  MoveL 696 to (-315.68, 55.52, -14.28) mm, rotated rx -179.9 ry 0 rz -90 deg; joints [13.027, -91.875, 133.091, -160.309, 41.97, 165.528]
  MoveL 697 to (-315.68, 55.53, -297.96) mm, rotated rx -179.9 ry 0 rz -90 deg; joints [10.215, -74.026, 113.034, -163.714, 39.206, 167.625]
  MoveC 698 to (-314.55, 55.52, -300.68) mm, rotated rx -179.9 ry 0 rz -90 deg; joints [10.243, -73.85, 112.805, -163.654, 39.161, 167.569] to (-311.82, 55.53, -301.81) mm, rotated rx -179.9 ry 0 rz -90 deg; joints [10.35, -73.753, 112.677, -163.476, 39.155, 167.427]
  MoveL 699 to (-311.82, 55.53, -301.81) mm, rotated rx -179.9 ry 0 rz -90 deg; joints [10.35, -73.753, 112.677, -163.476, 39.155, 167.427]
  MoveL 700 to (311.82, 55.52, -301.81) mm, rotated rx -179.9 ry 0 rz -90 deg; joints [33.565, -59.232, 91.443, -127.903, 44.47, 138.323]
  MoveC 701 to (314.55, 55.52, -300.68) mm, rotated rx -179.9 ry 0 rz -90 deg; joints [33.672, -59.197, 91.385, -127.772, 44.528, 138.219] to (315.68, 55.52, -297.96) mm, rotated rx -179.9 ry 0 rz -90 deg; joints [33.762, -59.301, 91.545, -127.721, 44.622, 138.214]
  MoveL 702 to (315.68, 55.53, -297.96) mm, rotated rx -179.9 ry 0 rz -90 deg; joints [33.762, -59.301, 91.545, -127.721, 44.622, 138.214]
  MoveL 703 to (315.68, 55.53, -141.98) mm, rotated rx -179.9 ry 0 rz -90 deg; joints [37.25, -67.192, 103.214, -126.934, 49.209, 139.929]
  MoveC 704 to (314.4, 55.52, -137.76) mm, rotated rx -179.9 ry 0 rz -90 deg; joints [37.312, -67.444, 103.572, -126.944, 49.312, 140] to (311, 55.53, -134.96) mm, rotated rx -179.9 ry 0 rz -90 deg; joints [37.272, -67.705, 103.944, -127.061, 49.353, 140.143]
  MoveL 705 to (311, 55.53, -134.96) mm, rotated rx -179.9 ry 0 rz -90 deg; joints [37.272, -67.705, 103.944, -127.061, 49.353, 140.143]
  MoveC 706 to (307.59, 55.53, -132.16) mm, rotated rx -179.9 ry 0 rz -90 deg; joints [37.231, -67.966, 104.315, -127.177, 49.393, 140.284] to (306.32, 55.52, -127.94) mm, rotated rx -179.9 ry 0 rz -90 deg; joints [37.294, -68.219, 104.669, -127.184, 49.495, 140.351]
  MoveL 707 to (306.31, 55.53, -127.94) mm, rotated rx -179.9 ry 0 rz -90 deg; joints [37.294, -68.219, 104.669, -127.184, 49.495, 140.351]
  MoveL 708 to (306.32, 55.53, -23.64) mm, rotated rx -179.9 ry 0 rz -90 deg; joints [40.023, -73.194, 111.401, -125.63, 52.284, 140.513]
  MoveC 709 to (305.19, 55.52, -20.92) mm, rotated rx -179.9 ry 0 rz -90 deg; joints [40.061, -73.365, 111.626, -125.627, 52.34, 140.546] to (302.46, 55.53, -19.79) mm, rotated rx -179.9 ry 0 rz -90 deg; joints [40.003, -73.525, 111.837, -125.716, 52.333, 140.633]
  MoveL 710 to (302.46, 55.52, -19.79) mm, rotated rx -179.9 ry 0 rz -90 deg; joints [40.003, -73.525, 111.837, -125.716, 52.333, 140.633]
  MoveL 711 to (-302.46, 55.52, -19.79) mm, rotated rx -179.9 ry 0 rz -90 deg; joints [13.666, -91.295, 132.533, -159.397, 42.156, 164.867]
  MoveC 712 to (-305.19, 55.53, -20.92) mm, rotated rx -179.9 ry 0 rz -90 deg; joints [13.506, -91.263, 132.504, -159.629, 42.117, 165.037] to (-306.32, 55.53, -23.64) mm, rotated rx -179.9 ry 0 rz -90 deg; joints [13.41, -91.098, 132.348, -159.769, 42.099, 165.141]
  MoveL 713 to (-306.31, 55.53, -23.64) mm, rotated rx -179.9 ry 0 rz -90 deg; joints [13.41, -91.098, 132.348, -159.769, 42.099, 165.141]
  MoveL 714 to (-306.32, 55.52, -288.59) mm, rotated rx -179.9 ry 0 rz -90 deg; joints [10.693, -74.485, 113.625, -163.024, 39.438, 167.123]
  MoveC 715 to (-305.19, 55.53, -291.32) mm, rotated rx -179.9 ry 0 rz -90 deg; joints [10.72, -74.309, 113.397, -162.965, 39.394, 167.068] to (-302.46, 55.52, -292.45) mm, rotated rx -179.9 ry 0 rz -90 deg; joints [10.827, -74.211, 113.268, -162.789, 39.39, 166.928]
  MoveL 716 to (-302.46, 55.52, -292.45) mm, rotated rx -179.9 ry 0 rz -90 deg; joints [10.827, -74.211, 113.268, -162.789, 39.39, 166.928]
  MoveL 717 to (302.46, 55.52, -292.45) mm, rotated rx -179.9 ry 0 rz -90 deg; joints [33.468, -60.052, 92.711, -128.364, 44.683, 138.897]
  MoveC 718 to (305.19, 55.53, -291.32) mm, rotated rx -179.9 ry 0 rz -90 deg; joints [33.576, -60.017, 92.655, -128.232, 44.741, 138.794] to (306.32, 55.53, -288.59) mm, rotated rx -179.9 ry 0 rz -90 deg; joints [33.667, -60.121, 92.813, -128.178, 44.834, 138.786]
  MoveL 719 to (306.31, 55.53, -288.59) mm, rotated rx -179.9 ry 0 rz -90 deg; joints [33.667, -60.121, 92.813, -128.178, 44.834, 138.786]
  MoveL 720 to (306.31, 55.53, -127.94) mm, rotated rx -179.9 ry 0 rz -90 deg; joints [37.294, -68.219, 104.669, -127.184, 49.495, 140.351]
  MoveC 721 to (305.04, 55.52, -123.72) mm, rotated rx -179.9 ry 0 rz -90 deg; joints [37.357, -68.47, 105.022, -127.189, 49.596, 140.417] to (301.63, 55.53, -120.92) mm, rotated rx -179.9 ry 0 rz -90 deg; joints [37.316, -68.731, 105.389, -127.302, 49.634, 140.554]
  MoveL 722 to (301.63, 55.52, -120.92) mm, rotated rx -179.9 ry 0 rz -90 deg; joints [37.316, -68.731, 105.389, -127.302, 49.634, 140.554]
  MoveC 723 to (298.23, 55.53, -118.11) mm, rotated rx -179.9 ry 0 rz -90 deg; joints [37.275, -68.992, 105.754, -127.414, 49.672, 140.689] to (296.95, 55.53, -113.9) mm, rotated rx -179.9 ry 0 rz -90 deg; joints [37.338, -69.244, 106.104, -127.415, 49.772, 140.751]
  MoveL 724 to (296.95, 55.53, -113.9) mm, rotated rx -179.9 ry 0 rz -90 deg; joints [37.338, -69.244, 106.104, -127.415, 49.772, 140.751]
  MoveL 725 to (296.95, 55.53, -33) mm, rotated rx -179.9 ry 0 rz -90 deg; joints [39.455, -73.116, 111.311, -126.178, 51.915, 140.832]
  MoveC 726 to (295.82, 55.53, -30.28) mm, rotated rx -179.9 ry 0 rz -90 deg; joints [39.492, -73.288, 111.537, -126.175, 51.971, 140.866] to (293.1, 55.52, -29.15) mm, rotated rx -179.9 ry 0 rz -90 deg; joints [39.433, -73.446, 111.747, -126.267, 51.964, 140.954]
  MoveL 727 to (293.1, 55.53, -29.15) mm, rotated rx -179.9 ry 0 rz -90 deg; joints [39.433, -73.446, 111.747, -126.267, 51.964, 140.954]
  MoveL 728 to (-293.1, 55.52, -29.15) mm, rotated rx -179.9 ry 0 rz -90 deg; joints [14.039, -90.518, 131.781, -158.872, 42.278, 164.489]
  MoveC 729 to (-295.82, 55.52, -30.28) mm, rotated rx -179.9 ry 0 rz -90 deg; joints [13.88, -90.488, 131.753, -159.1, 42.238, 164.656] to (-296.95, 55.52, -33) mm, rotated rx -179.9 ry 0 rz -90 deg; joints [13.785, -90.325, 131.595, -159.238, 42.218, 164.758]
  MoveL 730 to (-296.95, 55.53, -33) mm, rotated rx -179.9 ry 0 rz -90 deg; joints [13.785, -90.325, 131.595, -159.238, 42.218, 164.758]
  MoveL 731 to (-296.95, 55.52, -279.23) mm, rotated rx -179.9 ry 0 rz -90 deg; joints [11.177, -74.94, 114.205, -162.331, 39.669, 166.62]
  MoveC 732 to (-295.82, 55.52, -281.95) mm, rotated rx -179.9 ry 0 rz -90 deg; joints [11.202, -74.763, 113.978, -162.274, 39.627, 166.566] to (-293.1, 55.53, -283.08) mm, rotated rx -179.9 ry 0 rz -90 deg; joints [11.31, -74.664, 113.848, -162.098, 39.624, 166.427]
  MoveL 733 to (-293.1, 55.53, -283.08) mm, rotated rx -179.9 ry 0 rz -90 deg; joints [11.31, -74.664, 113.848, -162.098, 39.624, 166.427]
  MoveL 734 to (293.1, 55.53, -283.08) mm, rotated rx -179.9 ry 0 rz -90 deg; joints [33.37, -60.867, 93.962, -128.813, 44.89, 139.454]
  MoveC 735 to (295.82, 55.53, -281.95) mm, rotated rx -179.9 ry 0 rz -90 deg; joints [33.478, -60.832, 93.907, -128.68, 44.948, 139.351] to (296.95, 55.53, -279.23) mm, rotated rx -179.9 ry 0 rz -90 deg; joints [33.57, -60.936, 94.063, -128.623, 45.041, 139.341]
  MoveL 736 to (296.95, 55.52, -279.23) mm, rotated rx -179.9 ry 0 rz -90 deg; joints [33.57, -60.936, 94.063, -128.623, 45.041, 139.341]
  MoveL 737 to (296.95, 55.53, -113.9) mm, rotated rx -179.9 ry 0 rz -90 deg; joints [37.338, -69.244, 106.104, -127.415, 49.772, 140.751]
  MoveC 738 to (295.67, 55.53, -109.68) mm, rotated rx -179.9 ry 0 rz -90 deg; joints [37.402, -69.495, 106.452, -127.416, 49.871, 140.81] to (292.27, 55.53, -106.87) mm, rotated rx -179.9 ry 0 rz -90 deg; joints [37.361, -69.756, 106.814, -127.525, 49.906, 140.942]
  MoveL 739 to (292.27, 55.52, -106.87) mm, rotated rx -179.9 ry 0 rz -90 deg; joints [37.361, -69.756, 106.814, -127.525, 49.907, 140.942]
  MoveC 740 to (288.87, 55.52, -104.07) mm, rotated rx -179.9 ry 0 rz -90 deg; joints [37.32, -70.017, 107.175, -127.634, 49.941, 141.072] to (287.59, 55.52, -99.85) mm, rotated rx -179.9 ry 0 rz -90 deg; joints [37.384, -70.268, 107.519, -127.63, 50.039, 141.127]
  MoveL 741 to (287.59, 55.52, -99.85) mm, rotated rx -179.9 ry 0 rz -90 deg; joints [37.384, -70.268, 107.519, -127.63, 50.039, 141.127]
  MoveL 742 to (287.59, 55.52, -42.37) mm, rotated rx -179.9 ry 0 rz -90 deg; joints [38.888, -73.029, 111.21, -126.728, 51.549, 141.155]
  MoveC 743 to (286.46, 55.52, -39.64) mm, rotated rx -179.9 ry 0 rz -90 deg; joints [38.924, -73.202, 111.438, -126.727, 51.604, 141.189] to (283.74, 55.52, -38.51) mm, rotated rx -179.9 ry 0 rz -90 deg; joints [38.864, -73.359, 111.647, -126.82, 51.597, 141.279]
  MoveL 744 to (283.74, 55.52, -38.51) mm, rotated rx -179.9 ry 0 rz -90 deg; joints [38.864, -73.359, 111.647, -126.82, 51.597, 141.279]
  MoveL 745 to (-283.74, 55.53, -38.51) mm, rotated rx -179.9 ry 0 rz -90 deg; joints [14.404, -89.745, 131.019, -158.355, 42.389, 164.116]
  MoveC 746 to (-286.46, 55.52, -39.64) mm, rotated rx -179.9 ry 0 rz -90 deg; joints [14.247, -89.716, 130.992, -158.58, 42.348, 164.28] to (-287.59, 55.53, -42.37) mm, rotated rx -179.9 ry 0 rz -90 deg; joints [14.152, -89.555, 130.834, -158.716, 42.325, 164.38]
  MoveL 747 to (-287.59, 55.52, -42.37) mm, rotated rx -179.9 ry 0 rz -90 deg; joints [14.152, -89.555, 130.834, -158.716, 42.325, 164.38]
  MoveL 748 to (-287.59, 55.52, -269.87) mm, rotated rx -179.9 ry 0 rz -90 deg; joints [11.666, -75.39, 114.775, -161.634, 39.901, 166.115]
  MoveC 749 to (-286.46, 55.52, -272.59) mm, rotated rx -179.9 ry 0 rz -90 deg; joints [11.69, -75.213, 114.548, -161.578, 39.86, 166.063] to (-283.74, 55.52, -273.72) mm, rotated rx -179.9 ry 0 rz -90 deg; joints [11.798, -75.111, 114.417, -161.404, 39.858, 165.925]
  MoveL 750 to (-283.74, 55.52, -273.72) mm, rotated rx -179.9 ry 0 rz -90 deg; joints [11.798, -75.111, 114.417, -161.404, 39.858, 165.925]
  MoveL 751 to (283.74, 55.52, -273.72) mm, rotated rx -179.9 ry 0 rz -90 deg; joints [33.27, -61.677, 95.196, -129.25, 45.092, 139.994]
  MoveC 752 to (286.46, 55.52, -272.59) mm, rotated rx -179.9 ry 0 rz -90 deg; joints [33.379, -61.643, 95.142, -129.116, 45.15, 139.891] to (287.59, 55.52, -269.87) mm, rotated rx -179.9 ry 0 rz -90 deg; joints [33.472, -61.746, 95.296, -129.056, 45.242, 139.878]
  MoveL 753 to (287.59, 55.53, -269.87) mm, rotated rx -179.9 ry 0 rz -90 deg; joints [33.472, -61.746, 95.296, -129.056, 45.242, 139.878]
  MoveL 754 to (287.59, 55.52, -99.85) mm, rotated rx -179.9 ry 0 rz -90 deg; joints [37.384, -70.268, 107.519, -127.63, 50.039, 141.127]
  MoveC 755 to (286.31, 55.53, -95.63) mm, rotated rx -179.9 ry 0 rz -90 deg; joints [37.449, -70.519, 107.863, -127.626, 50.136, 141.181] to (282.91, 55.52, -92.83) mm, rotated rx -179.9 ry 0 rz -90 deg; joints [37.407, -70.78, 108.22, -127.732, 50.169, 141.307]
  MoveL 756 to (282.91, 55.52, -92.83) mm, rotated rx -179.9 ry 0 rz -90 deg; joints [37.407, -70.78, 108.22, -127.732, 50.169, 141.307]
  MoveC 757 to (279.5, 55.52, -90.03) mm, rotated rx -179.9 ry 0 rz -90 deg; joints [37.366, -71.041, 108.576, -127.837, 50.201, 141.432] to (278.23, 55.52, -85.81) mm, rotated rx -179.9 ry 0 rz -90 deg; joints [37.431, -71.292, 108.916, -127.829, 50.296, 141.481]
  MoveL 758 to (278.23, 55.53, -85.81) mm, rotated rx -179.9 ry 0 rz -90 deg; joints [37.431, -71.292, 108.916, -127.829, 50.296, 141.481]
  MoveL 759 to (278.23, 55.53, -51.73) mm, rotated rx -179.9 ry 0 rz -90 deg; joints [38.323, -72.935, 111.099, -127.28, 51.183, 141.48]
  MoveC 760 to (277.1, 55.53, -49.01) mm, rotated rx -179.9 ry 0 rz -90 deg; joints [38.357, -73.108, 111.327, -127.281, 51.238, 141.515] to (274.37, 55.52, -47.88) mm, rotated rx -179.9 ry 0 rz -90 deg; joints [38.296, -73.265, 111.535, -127.376, 51.231, 141.605]
  MoveL 761 to (274.37, 55.52, -47.88) mm, rotated rx -179.9 ry 0 rz -90 deg; joints [38.296, -73.265, 111.535, -127.376, 51.231, 141.605]
  MoveL 762 to (-274.37, 55.52, -47.88) mm, rotated rx -179.9 ry 0 rz -90 deg; joints [14.762, -88.975, 130.248, -157.846, 42.489, 163.746]
  MoveC 763 to (-277.1, 55.52, -49.01) mm, rotated rx -179.9 ry 0 rz -90 deg; joints [14.606, -88.947, 130.222, -158.068, 42.447, 163.908] to (-278.23, 55.52, -51.73) mm, rotated rx -179.9 ry 0 rz -90 deg; joints [14.512, -88.789, 130.064, -158.202, 42.42, 164.005]
  MoveL 764 to (-278.23, 55.52, -51.73) mm, rotated rx -179.9 ry 0 rz -90 deg; joints [14.512, -88.789, 130.064, -158.202, 42.42, 164.005]
  MoveL 765 to (-278.23, 55.52, -260.51) mm, rotated rx -179.9 ry 0 rz -90 deg; joints [12.16, -75.835, 115.335, -160.932, 40.132, 165.61]
  MoveC 766 to (-277.1, 55.52, -263.23) mm, rotated rx -179.9 ry 0 rz -90 deg; joints [12.184, -75.657, 115.109, -160.879, 40.092, 165.559] to (-274.37, 55.52, -264.36) mm, rotated rx -179.9 ry 0 rz -90 deg; joints [12.292, -75.554, 114.977, -160.705, 40.092, 165.422]
  MoveL 767 to (-274.37, 55.52, -264.36) mm, rotated rx -179.9 ry 0 rz -90 deg; joints [12.292, -75.554, 114.977, -160.705, 40.092, 165.422]
  MoveL 768 to (274.37, 55.52, -264.36) mm, rotated rx -179.9 ry 0 rz -90 deg; joints [33.168, -62.482, 96.413, -129.675, 45.289, 140.518]
  MoveC 769 to (277.1, 55.52, -263.23) mm, rotated rx -179.9 ry 0 rz -90 deg; joints [33.279, -62.449, 96.36, -129.541, 45.347, 140.415] to (278.23, 55.52, -260.51) mm, rotated rx -179.9 ry 0 rz -90 deg; joints [33.372, -62.552, 96.513, -129.479, 45.438, 140.4]
  MoveL 770 to (278.23, 55.52, -260.51) mm, rotated rx -179.9 ry 0 rz -90 deg; joints [33.372, -62.552, 96.513, -129.479, 45.438, 140.4]
  MoveL 771 to (278.23, 55.53, -85.81) mm, rotated rx -179.9 ry 0 rz -90 deg; joints [37.431, -71.292, 108.916, -127.829, 50.296, 141.481]
  MoveC 772 to (276.95, 55.52, -81.59) mm, rotated rx -179.9 ry 0 rz -90 deg; joints [37.497, -71.544, 109.255, -127.819, 50.391, 141.529] to (273.55, 55.52, -78.79) mm, rotated rx -179.9 ry 0 rz -90 deg; joints [37.455, -71.805, 109.608, -127.922, 50.421, 141.65]
  MoveL 773 to (273.55, 55.52, -78.79) mm, rotated rx -179.9 ry 0 rz -90 deg; joints [37.455, -71.805, 109.608, -127.922, 50.421, 141.65]
  MoveC 774 to (270.14, 55.52, -75.98) mm, rotated rx -179.9 ry 0 rz -90 deg; joints [37.413, -72.065, 109.959, -128.024, 50.451, 141.769] to (268.86, 55.53, -71.76) mm, rotated rx -179.9 ry 0 rz -90 deg; joints [37.479, -72.317, 110.295, -128.011, 50.544, 141.813]
  MoveL 775 to (268.86, 55.53, -71.76) mm, rotated rx -179.9 ry 0 rz -90 deg; joints [37.479, -72.317, 110.295, -128.011, 50.544, 141.813]
  MoveL 776 to (268.86, 55.52, -61.09) mm, rotated rx -179.9 ry 0 rz -90 deg; joints [37.758, -72.834, 110.977, -127.835, 50.819, 141.807]
  MoveC 777 to (267.74, 55.53, -58.37) mm, rotated rx -179.9 ry 0 rz -90 deg; joints [37.792, -73.007, 111.206, -127.837, 50.874, 141.843] to (265.01, 55.53, -57.24) mm, rotated rx -179.9 ry 0 rz -90 deg; joints [37.729, -73.163, 111.413, -127.934, 50.867, 141.935]
  MoveL 778 to (265.01, 55.52, -57.24) mm, rotated rx -179.9 ry 0 rz -90 deg; joints [37.729, -73.163, 111.413, -127.934, 50.867, 141.935]
  MoveL 779 to (-265.01, 55.53, -57.24) mm, rotated rx -179.9 ry 0 rz -90 deg; joints [15.112, -88.208, 129.468, -157.345, 42.577, 163.379]
  MoveC 780 to (-267.74, 55.52, -58.37) mm, rotated rx -179.9 ry 0 rz -90 deg; joints [14.958, -88.182, 129.443, -157.563, 42.534, 163.538] to (-268.86, 55.53, -61.09) mm, rotated rx -179.9 ry 0 rz -90 deg; joints [14.863, -88.025, 129.284, -157.696, 42.505, 163.634]
  MoveL 781 to (-268.86, 55.52, -61.09) mm, rotated rx -179.9 ry 0 rz -90 deg; joints [14.863, -88.025, 129.284, -157.696, 42.505, 163.634]
  MoveL 782 to (-268.86, 55.52, -251.14) mm, rotated rx -179.9 ry 0 rz -90 deg; joints [12.661, -76.274, 115.884, -160.227, 40.363, 165.104]
  MoveC 783 to (-267.74, 55.53, -253.87) mm, rotated rx -179.9 ry 0 rz -90 deg; joints [12.683, -76.096, 115.658, -160.175, 40.325, 165.054] to (-265.01, 55.52, -255) mm, rotated rx -179.9 ry 0 rz -90 deg; joints [12.791, -75.992, 115.525, -160.003, 40.326, 164.918]
  MoveL 784 to (-265.01, 55.53, -255) mm, rotated rx -179.9 ry 0 rz -90 deg; joints [12.791, -75.992, 115.525, -160.003, 40.326, 164.918]
  MoveL 785 to (265.01, 55.52, -255) mm, rotated rx -179.9 ry 0 rz -90 deg; joints [33.065, -63.284, 97.615, -130.09, 45.479, 141.026]
  MoveC 786 to (267.74, 55.52, -253.87) mm, rotated rx -179.9 ry 0 rz -90 deg; joints [33.176, -63.251, 97.563, -129.955, 45.538, 140.923] to (268.86, 55.52, -251.14) mm, rotated rx -179.9 ry 0 rz -90 deg; joints [33.27, -63.354, 97.714, -129.89, 45.628, 140.906]
  MoveL 787 to (268.86, 55.52, -251.14) mm, rotated rx -179.9 ry 0 rz -90 deg; joints [33.27, -63.354, 97.714, -129.89, 45.628, 140.906]
  MoveL 788 to (268.86, 55.53, -71.76) mm, rotated rx -179.9 ry 0 rz -90 deg; joints [37.479, -72.317, 110.295, -128.011, 50.544, 141.813]
  MoveC 789 to (266.09, 55.52, -66.2) mm, rotated rx -179.9 ry 0 rz -90 deg; joints [37.53, -72.689, 110.789, -128.038, 50.651, 141.906] to (259.98, 55.53, -65.06) mm, rotated rx -179.9 ry 0 rz -90 deg; joints [37.352, -72.969, 111.165, -128.281, 50.601, 142.116]
  MoveL 790 to (259.98, 55.53, -65.06) mm, rotated rx -179.9 ry 0 rz -90 deg; joints [37.352, -72.969, 111.165, -128.281, 50.601, 142.116]
  MoveC 791 to (254.53, 55.52, -66.22) mm, rotated rx -179.9 ry 0 rz -90 deg; joints [37.136, -73.112, 111.361, -128.536, 50.499, 142.305] to (248.97, 55.53, -66.6) mm, rotated rx -179.9 ry 0 rz -90 deg; joints [36.934, -73.296, 111.608, -128.783, 50.416, 142.498]
  MoveL 792 to (248.97, 55.53, -66.6) mm, rotated rx -179.9 ry 0 rz -90 deg; joints [36.934, -73.296, 111.608, -128.783, 50.416, 142.498]
  MoveL 793 to (-255.65, 55.53, -66.6) mm, rotated rx -179.9 ry 0 rz -90 deg; joints [15.454, -87.444, 128.679, -156.85, 42.654, 163.014]
  MoveC 794 to (-258.37, 55.53, -67.73) mm, rotated rx -179.9 ry 0 rz -90 deg; joints [15.302, -87.42, 128.656, -157.066, 42.61, 163.171] to (-259.5, 55.52, -70.46) mm, rotated rx -179.9 ry 0 rz -90 deg; joints [15.208, -87.265, 128.496, -157.197, 42.578, 163.264]
  MoveL 795 to (-259.5, 55.52, -70.46) mm, rotated rx -179.9 ry 0 rz -90 deg; joints [15.208, -87.265, 128.496, -157.197, 42.578, 163.264]
  MoveL 796 to (-259.5, 55.52, -241.78) mm, rotated rx -179.9 ry 0 rz -90 deg; joints [13.166, -76.708, 116.422, -159.518, 40.595, 164.596]
  MoveC 797 to (-258.37, 55.53, -244.5) mm, rotated rx -179.9 ry 0 rz -90 deg; joints [13.188, -76.529, 116.198, -159.468, 40.558, 164.548] to (-255.65, 55.53, -245.63) mm, rotated rx -179.9 ry 0 rz -90 deg; joints [13.295, -76.424, 116.064, -159.297, 40.561, 164.413]
  MoveL 798 to (-255.65, 55.53, -245.63) mm, rotated rx -179.9 ry 0 rz -90 deg; joints [13.295, -76.424, 116.064, -159.297, 40.561, 164.413]
  MoveL 799 to (255.65, 55.52, -245.63) mm, rotated rx -179.9 ry 0 rz -90 deg; joints [32.959, -64.082, 98.801, -130.495, 45.664, 141.519]
  MoveC 800 to (258.37, 55.53, -244.5) mm, rotated rx -179.9 ry 0 rz -90 deg; joints [33.072, -64.05, 98.751, -130.359, 45.723, 141.416] to (259.5, 55.52, -241.78) mm, rotated rx -179.9 ry 0 rz -90 deg; joints [33.166, -64.153, 98.901, -130.291, 45.812, 141.396]
  MoveL 801 to (259.5, 55.52, -241.78) mm, rotated rx -179.9 ry 0 rz -90 deg; joints [33.166, -64.153, 98.901, -130.291, 45.812, 141.396]
  MoveL 802 to (259.5, 55.53, -70.46) mm, rotated rx -179.9 ry 0 rz -90 deg; joints [37.195, -72.724, 110.844, -128.392, 50.456, 142.137]
  MoveC 803 to (258.37, 55.53, -67.73) mm, rotated rx -179.9 ry 0 rz -90 deg; joints [37.228, -72.898, 111.074, -128.395, 50.511, 142.174] to (255.65, 55.52, -66.6) mm, rotated rx -179.9 ry 0 rz -90 deg; joints [37.164, -73.052, 111.281, -128.494, 50.504, 142.267]
  MoveL 804 to (255.65, 55.52, -66.6) mm, rotated rx -179.9 ry 0 rz -90 deg; joints [37.164, -73.052, 111.281, -128.494, 50.504, 142.267]
  MoveL 805 to (248.97, 55.53, -66.6) mm, rotated rx -179.9 ry 0 rz -90 deg; joints [36.934, -73.296, 111.608, -128.783, 50.416, 142.498]
  MoveC 806 to (244.46, 55.52, -67.86) mm, rotated rx -179.9 ry 0 rz -90 deg; joints [36.746, -73.398, 111.746, -129, 50.324, 142.655] to (241.27, 55.52, -71.28) mm, rotated rx -179.9 ry 0 rz -90 deg; joints [36.547, -73.345, 111.682, -129.197, 50.195, 142.771]
  MoveL 807 to (241.27, 55.52, -71.28) mm, rotated rx -179.9 ry 0 rz -90 deg; joints [36.547, -73.345, 111.682, -129.197, 50.195, 142.771]
  MoveC 808 to (238.08, 55.52, -74.7) mm, rotated rx -179.9 ry 0 rz -90 deg; joints [36.349, -73.292, 111.616, -129.395, 50.067, 142.886] to (233.58, 55.53, -75.96) mm, rotated rx -179.9 ry 0 rz -90 deg; joints [36.16, -73.391, 111.75, -129.614, 49.975, 143.046]
  MoveL 809 to (233.58, 55.53, -75.96) mm, rotated rx -179.9 ry 0 rz -90 deg; joints [36.16, -73.391, 111.75, -129.614, 49.975, 143.046]
  MoveL 810 to (-246.29, 55.53, -75.96) mm, rotated rx -179.9 ry 0 rz -90 deg; joints [15.79, -86.684, 127.882, -156.362, 42.721, 162.651]
  MoveC 811 to (-249.01, 55.53, -77.09) mm, rotated rx -179.9 ry 0 rz -90 deg; joints [15.639, -86.66, 127.859, -156.575, 42.676, 162.805] to (-250.14, 55.52, -79.82) mm, rotated rx -179.9 ry 0 rz -90 deg; joints [15.545, -86.507, 127.699, -156.704, 42.641, 162.896]
  MoveL 812 to (-250.14, 55.53, -79.82) mm, rotated rx -179.9 ry 0 rz -90 deg; joints [15.545, -86.507, 127.699, -156.704, 42.641, 162.896]
  MoveL 813 to (-250.14, 55.52, -232.42) mm, rotated rx -179.9 ry 0 rz -90 deg; joints [13.677, -77.137, 116.95, -158.806, 40.828, 164.087]
  MoveC 814 to (-249.01, 55.53, -235.14) mm, rotated rx -179.9 ry 0 rz -90 deg; joints [13.698, -76.958, 116.727, -158.757, 40.792, 164.04] to (-246.29, 55.52, -236.27) mm, rotated rx -179.9 ry 0 rz -90 deg; joints [13.805, -76.851, 116.592, -158.588, 40.796, 163.907]
  MoveL 815 to (-246.29, 55.53, -236.27) mm, rotated rx -179.9 ry 0 rz -90 deg; joints [13.805, -76.851, 116.592, -158.588, 40.796, 163.907]
  MoveL 816 to (246.29, 55.53, -236.27) mm, rotated rx -179.9 ry 0 rz -90 deg; joints [32.852, -64.878, 99.973, -130.89, 45.843, 141.998]
  MoveC 817 to (249.01, 55.53, -235.14) mm, rotated rx -179.9 ry 0 rz -90 deg; joints [32.966, -64.846, 99.924, -130.754, 45.902, 141.895] to (250.14, 55.52, -232.42) mm, rotated rx -179.9 ry 0 rz -90 deg; joints [33.061, -64.949, 100.072, -130.683, 45.99, 141.873]
  MoveL 818 to (250.14, 55.53, -232.42) mm, rotated rx -179.9 ry 0 rz -90 deg; joints [33.061, -64.949, 100.072, -130.683, 45.99, 141.873]
  MoveL 819 to (250.14, 55.53, -79.82) mm, rotated rx -179.9 ry 0 rz -90 deg; joints [36.634, -72.607, 110.701, -128.951, 50.095, 142.47]
  MoveC 820 to (249.01, 55.53, -77.09) mm, rotated rx -179.9 ry 0 rz -90 deg; joints [36.665, -72.781, 110.932, -128.956, 50.15, 142.508] to (246.29, 55.53, -75.96) mm, rotated rx -179.9 ry 0 rz -90 deg; joints [36.6, -72.935, 111.137, -129.056, 50.143, 142.602]
  MoveL 821 to (246.29, 55.52, -75.96) mm, rotated rx -179.9 ry 0 rz -90 deg; joints [36.6, -72.934, 111.137, -129.056, 50.143, 142.602]
  MoveL 822 to (233.58, 55.53, -75.96) mm, rotated rx -179.9 ry 0 rz -90 deg; joints [36.16, -73.391, 111.75, -129.614, 49.975, 143.046]
  MoveC 823 to (229.36, 55.52, -77.24) mm, rotated rx -179.9 ry 0 rz -90 deg; joints [35.98, -73.478, 111.869, -129.822, 49.887, 143.195] to (226.56, 55.52, -80.65) mm, rotated rx -179.9 ry 0 rz -90 deg; joints [35.795, -73.409, 111.782, -130.003, 49.765, 143.299]
  MoveL 824 to (226.56, 55.52, -80.65) mm, rotated rx -179.9 ry 0 rz -90 deg; joints [35.795, -73.409, 111.782, -130.003, 49.765, 143.299]
  MoveC 825 to (223.75, 55.53, -84.05) mm, rotated rx -179.9 ry 0 rz -90 deg; joints [35.611, -73.338, 111.694, -130.185, 49.642, 143.403] to (219.54, 55.53, -85.33) mm, rotated rx -179.9 ry 0 rz -90 deg; joints [35.431, -73.423, 111.81, -130.395, 49.555, 143.554]
  MoveL 826 to (219.54, 55.53, -85.33) mm, rotated rx -179.9 ry 0 rz -90 deg; joints [35.431, -73.423, 111.81, -130.395, 49.555, 143.554]
  MoveL 827 to (-236.92, 55.52, -85.33) mm, rotated rx -179.9 ry 0 rz -90 deg; joints [16.119, -85.926, 127.075, -155.88, 42.776, 162.289]
  MoveC 828 to (-239.65, 55.53, -86.46) mm, rotated rx -179.9 ry 0 rz -90 deg; joints [15.969, -85.904, 127.053, -156.089, 42.731, 162.44] to (-240.78, 55.52, -89.18) mm, rotated rx -179.9 ry 0 rz -90 deg; joints [15.876, -85.753, 126.893, -156.217, 42.694, 162.53]
  MoveL 829 to (-240.78, 55.52, -89.18) mm, rotated rx -179.9 ry 0 rz -90 deg; joints [15.876, -85.753, 126.893, -156.217, 42.694, 162.53]
  MoveL 830 to (-240.78, 55.52, -223.05) mm, rotated rx -179.9 ry 0 rz -90 deg; joints [14.194, -77.561, 117.468, -158.089, 41.061, 163.577]
  MoveC 831 to (-239.65, 55.52, -225.78) mm, rotated rx -179.9 ry 0 rz -90 deg; joints [14.213, -77.381, 117.245, -158.043, 41.027, 163.532] to (-236.92, 55.52, -226.91) mm, rotated rx -179.9 ry 0 rz -90 deg; joints [14.321, -77.272, 117.109, -157.874, 41.033, 163.4]
  MoveL 832 to (-236.92, 55.52, -226.91) mm, rotated rx -179.9 ry 0 rz -90 deg; joints [14.321, -77.272, 117.109, -157.874, 41.033, 163.4]
  MoveL 833 to (236.92, 55.52, -226.91) mm, rotated rx -179.9 ry 0 rz -90 deg; joints [32.743, -65.671, 101.131, -131.277, 46.016, 142.463]
  MoveC 834 to (239.65, 55.53, -225.78) mm, rotated rx -179.9 ry 0 rz -90 deg; joints [32.857, -65.639, 101.083, -131.139, 46.075, 142.36] to (240.78, 55.53, -223.05) mm, rotated rx -179.9 ry 0 rz -90 deg; joints [32.953, -65.742, 101.23, -131.066, 46.163, 142.335]
  MoveL 835 to (240.78, 55.53, -223.05) mm, rotated rx -179.9 ry 0 rz -90 deg; joints [32.953, -65.742, 101.23, -131.066, 46.163, 142.335]
  MoveL 836 to (240.78, 55.53, -89.18) mm, rotated rx -179.9 ry 0 rz -90 deg; joints [36.074, -72.481, 110.547, -129.512, 49.736, 142.805]
  MoveC 837 to (239.65, 55.52, -86.46) mm, rotated rx -179.9 ry 0 rz -90 deg; joints [36.104, -72.656, 110.779, -129.518, 49.79, 142.843] to (236.92, 55.52, -85.33) mm, rotated rx -179.9 ry 0 rz -90 deg; joints [36.038, -72.809, 110.984, -129.621, 49.783, 142.939]
  MoveL 838 to (236.92, 55.52, -85.33) mm, rotated rx -179.9 ry 0 rz -90 deg; joints [36.038, -72.809, 110.984, -129.621, 49.783, 142.939]
  MoveL 839 to (219.54, 55.53, -85.33) mm, rotated rx -179.9 ry 0 rz -90 deg; joints [35.431, -73.423, 111.81, -130.395, 49.555, 143.554]
  MoveC 840 to (215.32, 55.52, -86.61) mm, rotated rx -179.9 ry 0 rz -90 deg; joints [35.25, -73.507, 111.924, -130.605, 49.467, 143.705] to (212.51, 55.52, -90.01) mm, rotated rx -179.9 ry 0 rz -90 deg; joints [35.066, -73.435, 111.833, -130.788, 49.345, 143.81]
  MoveL 841 to (212.51, 55.52, -90.01) mm, rotated rx -179.9 ry 0 rz -90 deg; joints [35.066, -73.435, 111.833, -130.788, 49.345, 143.81]
  MoveC 842 to (209.71, 55.53, -93.41) mm, rotated rx -179.9 ry 0 rz -90 deg; joints [34.883, -73.361, 111.74, -130.97, 49.224, 143.915] to (205.49, 55.53, -94.69) mm, rotated rx -179.9 ry 0 rz -90 deg; joints [34.701, -73.443, 111.852, -131.183, 49.136, 144.068]
  MoveL 843 to (205.49, 55.53, -94.69) mm, rotated rx -179.9 ry 0 rz -90 deg; joints [34.701, -73.443, 111.852, -131.183, 49.136, 144.068]
  MoveL 844 to (-227.56, 55.52, -94.69) mm, rotated rx -179.9 ry 0 rz -90 deg; joints [16.44, -85.171, 126.26, -155.403, 42.821, 161.927]
  MoveC 845 to (-230.29, 55.52, -95.82) mm, rotated rx -179.9 ry 0 rz -90 deg; joints [16.292, -85.15, 126.239, -155.61, 42.775, 162.076] to (-231.41, 55.53, -98.54) mm, rotated rx -179.9 ry 0 rz -90 deg; joints [16.199, -85, 126.078, -155.735, 42.736, 162.164]
  MoveL 846 to (-231.41, 55.52, -98.54) mm, rotated rx -179.9 ry 0 rz -90 deg; joints [16.199, -85, 126.078, -155.735, 42.736, 162.164]
  MoveL 847 to (-231.41, 55.53, -213.69) mm, rotated rx -179.9 ry 0 rz -90 deg; joints [14.717, -77.979, 117.976, -157.369, 41.296, 163.065]
  MoveC 848 to (-230.29, 55.52, -216.42) mm, rotated rx -179.9 ry 0 rz -90 deg; joints [14.735, -77.798, 117.753, -157.324, 41.263, 163.022] to (-227.56, 55.52, -217.54) mm, rotated rx -179.9 ry 0 rz -90 deg; joints [14.842, -77.688, 117.616, -157.157, 41.27, 162.891]
  MoveL 849 to (-227.56, 55.53, -217.55) mm, rotated rx -179.9 ry 0 rz -90 deg; joints [14.842, -77.688, 117.616, -157.157, 41.27, 162.891]
  MoveL 850 to (227.56, 55.53, -217.55) mm, rotated rx -179.9 ry 0 rz -90 deg; joints [32.632, -66.461, 102.275, -131.654, 46.182, 142.914]
  MoveC 851 to (230.29, 55.52, -216.42) mm, rotated rx -179.9 ry 0 rz -90 deg; joints [32.747, -66.43, 102.228, -131.515, 46.242, 142.811] to (231.41, 55.52, -213.69) mm, rotated rx -179.9 ry 0 rz -90 deg; joints [32.844, -66.533, 102.374, -131.44, 46.329, 142.784]
  MoveL 852 to (231.41, 55.52, -213.69) mm, rotated rx -179.9 ry 0 rz -90 deg; joints [32.844, -66.533, 102.374, -131.44, 46.329, 142.784]
  MoveL 853 to (231.41, 55.52, -98.54) mm, rotated rx -179.9 ry 0 rz -90 deg; joints [35.516, -72.349, 110.382, -130.075, 49.378, 143.142]
  MoveC 854 to (230.29, 55.52, -95.82) mm, rotated rx -179.9 ry 0 rz -90 deg; joints [35.544, -72.524, 110.615, -130.083, 49.432, 143.182] to (227.56, 55.53, -94.69) mm, rotated rx -179.9 ry 0 rz -90 deg; joints [35.478, -72.675, 110.819, -130.187, 49.425, 143.279]
  MoveL 855 to (227.56, 55.52, -94.69) mm, rotated rx -179.9 ry 0 rz -90 deg; joints [35.478, -72.675, 110.819, -130.187, 49.425, 143.279]
  MoveL 856 to (205.49, 55.53, -94.69) mm, rotated rx -179.9 ry 0 rz -90 deg; joints [34.701, -73.443, 111.852, -131.183, 49.136, 144.068]
  MoveC 857 to (201.27, 55.53, -95.97) mm, rotated rx -179.9 ry 0 rz -90 deg; joints [34.52, -73.524, 111.962, -131.396, 49.049, 144.222] to (198.47, 55.53, -99.37) mm, rotated rx -179.9 ry 0 rz -90 deg; joints [34.336, -73.448, 111.866, -131.58, 48.928, 144.328]
  MoveL 858 to (198.47, 55.52, -99.37) mm, rotated rx -179.9 ry 0 rz -90 deg; joints [34.336, -73.448, 111.866, -131.58, 48.928, 144.328]
  MoveC 859 to (195.67, 55.53, -102.78) mm, rotated rx -179.9 ry 0 rz -90 deg; joints [34.153, -73.371, 111.769, -131.764, 48.808, 144.435] to (191.45, 55.52, -104.05) mm, rotated rx -179.9 ry 0 rz -90 deg; joints [33.971, -73.449, 111.877, -131.979, 48.721, 144.59]
  MoveL 860 to (191.45, 55.52, -104.05) mm, rotated rx -179.9 ry 0 rz -90 deg; joints [33.971, -73.449, 111.877, -131.979, 48.721, 144.59]
  MoveL 861 to (-218.2, 55.53, -104.05) mm, rotated rx -179.9 ry 0 rz -90 deg; joints [16.756, -84.418, 125.435, -154.93, 42.856, 161.565]
  MoveC 862 to (-220.92, 55.53, -105.18) mm, rotated rx -179.9 ry 0 rz -90 deg; joints [16.609, -84.398, 125.415, -155.134, 42.809, 161.712] to (-222.05, 55.53, -107.91) mm, rotated rx -179.9 ry 0 rz -90 deg; joints [16.516, -84.25, 125.254, -155.258, 42.767, 161.798]
  MoveL 863 to (-222.05, 55.52, -107.91) mm, rotated rx -179.9 ry 0 rz -90 deg; joints [16.516, -84.25, 125.254, -155.258, 42.767, 161.798]
  MoveL 864 to (-222.05, 55.52, -204.33) mm, rotated rx -179.9 ry 0 rz -90 deg; joints [15.245, -78.391, 118.473, -156.645, 41.532, 162.553]
  MoveC 865 to (-220.92, 55.52, -207.05) mm, rotated rx -179.9 ry 0 rz -90 deg; joints [15.262, -78.21, 118.251, -156.602, 41.5, 162.511] to (-218.2, 55.53, -208.18) mm, rotated rx -179.9 ry 0 rz -90 deg; joints [15.369, -78.098, 118.113, -156.437, 41.508, 162.382]
  MoveL 866 to (-218.2, 55.53, -208.18) mm, rotated rx -179.9 ry 0 rz -90 deg; joints [15.369, -78.098, 118.113, -156.437, 41.508, 162.382]
  MoveL 867 to (218.2, 55.52, -208.18) mm, rotated rx -179.9 ry 0 rz -90 deg; joints [32.519, -67.249, 103.406, -132.023, 46.343, 143.352]
  MoveC 868 to (220.92, 55.53, -207.05) mm, rotated rx -179.9 ry 0 rz -90 deg; joints [32.635, -67.218, 103.36, -131.884, 46.402, 143.249] to (222.05, 55.52, -204.33) mm, rotated rx -179.9 ry 0 rz -90 deg; joints [32.733, -67.322, 103.505, -131.806, 46.489, 143.219]
  MoveL 869 to (222.05, 55.52, -204.33) mm, rotated rx -179.9 ry 0 rz -90 deg; joints [32.733, -67.322, 103.505, -131.806, 46.489, 143.219]
  MoveL 870 to (222.05, 55.53, -107.91) mm, rotated rx -179.9 ry 0 rz -90 deg; joints [34.959, -72.208, 110.207, -130.64, 49.021, 143.482]
  MoveC 871 to (220.92, 55.53, -105.18) mm, rotated rx -179.9 ry 0 rz -90 deg; joints [34.987, -72.384, 110.441, -130.649, 49.075, 143.523] to (218.2, 55.53, -104.05) mm, rotated rx -179.9 ry 0 rz -90 deg; joints [34.919, -72.534, 110.644, -130.755, 49.069, 143.621]
  MoveL 872 to (218.2, 55.53, -104.05) mm, rotated rx -179.9 ry 0 rz -90 deg; joints [34.919, -72.534, 110.644, -130.755, 49.069, 143.621]
  MoveL 873 to (191.45, 55.52, -104.05) mm, rotated rx -179.9 ry 0 rz -90 deg; joints [33.971, -73.449, 111.877, -131.979, 48.721, 144.59]
  MoveC 874 to (187.23, 55.52, -105.33) mm, rotated rx -179.9 ry 0 rz -90 deg; joints [33.789, -73.527, 111.982, -132.195, 48.634, 144.745] to (184.43, 55.52, -108.73) mm, rotated rx -179.9 ry 0 rz -90 deg; joints [33.606, -73.448, 111.882, -132.38, 48.514, 144.853]
  MoveL 875 to (184.43, 55.53, -108.73) mm, rotated rx -179.9 ry 0 rz -90 deg; joints [33.606, -73.448, 111.882, -132.38, 48.514, 144.853]
  MoveC 876 to (181.62, 55.52, -112.14) mm, rotated rx -179.9 ry 0 rz -90 deg; joints [33.424, -73.368, 111.781, -132.565, 48.394, 144.961] to (177.4, 55.52, -113.42) mm, rotated rx -179.9 ry 0 rz -90 deg; joints [33.241, -73.443, 111.884, -132.783, 48.307, 145.118]
  MoveL 877 to (177.4, 55.53, -113.42) mm, rotated rx -179.9 ry 0 rz -90 deg; joints [33.241, -73.443, 111.884, -132.783, 48.307, 145.118]
  MoveL 878 to (-208.84, 55.53, -113.42) mm, rotated rx -179.9 ry 0 rz -90 deg; joints [17.065, -83.668, 124.602, -154.462, 42.88, 161.203]
  MoveC 879 to (-211.56, 55.52, -114.54) mm, rotated rx -179.9 ry 0 rz -90 deg; joints [16.92, -83.649, 124.583, -154.664, 42.833, 161.348] to (-212.69, 55.53, -117.27) mm, rotated rx -179.9 ry 0 rz -90 deg; joints [16.827, -83.503, 124.421, -154.785, 42.789, 161.431]
  MoveL 880 to (-212.69, 55.53, -117.27) mm, rotated rx -179.9 ry 0 rz -90 deg; joints [16.827, -83.503, 124.421, -154.785, 42.789, 161.431]
  MoveL 881 to (-212.69, 55.53, -194.97) mm, rotated rx -179.9 ry 0 rz -90 deg; joints [15.778, -78.798, 118.959, -155.917, 41.769, 162.039]
  MoveC 882 to (-211.56, 55.52, -197.69) mm, rotated rx -179.9 ry 0 rz -90 deg; joints [15.794, -78.616, 118.739, -155.877, 41.739, 161.999] to (-208.84, 55.53, -198.82) mm, rotated rx -179.9 ry 0 rz -90 deg; joints [15.901, -78.503, 118.6, -155.712, 41.748, 161.871]
  MoveL 883 to (-208.84, 55.52, -198.82) mm, rotated rx -179.9 ry 0 rz -90 deg; joints [15.901, -78.503, 118.6, -155.712, 41.748, 161.871]
  MoveL 884 to (208.84, 55.53, -198.82) mm, rotated rx -179.9 ry 0 rz -90 deg; joints [32.404, -68.036, 104.525, -132.385, 46.497, 143.777]
  MoveC 885 to (211.56, 55.52, -197.69) mm, rotated rx -179.9 ry 0 rz -90 deg; joints [32.521, -68.006, 104.479, -132.244, 46.557, 143.674] to (212.69, 55.52, -194.97) mm, rotated rx -179.9 ry 0 rz -90 deg; joints [32.62, -68.109, 104.623, -132.164, 46.642, 143.642]
  MoveL 886 to (212.69, 55.53, -194.97) mm, rotated rx -179.9 ry 0 rz -90 deg; joints [32.62, -68.109, 104.623, -132.164, 46.642, 143.642]
  MoveL 887 to (212.69, 55.53, -117.27) mm, rotated rx -179.9 ry 0 rz -90 deg; joints [34.405, -72.06, 110.021, -131.206, 48.666, 143.825]
  MoveC 888 to (211.56, 55.52, -114.54) mm, rotated rx -179.9 ry 0 rz -90 deg; joints [34.431, -72.236, 110.256, -131.217, 48.72, 143.866] to (208.84, 55.52, -113.42) mm, rotated rx -179.9 ry 0 rz -90 deg; joints [34.363, -72.386, 110.458, -131.325, 48.714, 143.965]
  MoveL 889 to (208.84, 55.53, -113.42) mm, rotated rx -179.9 ry 0 rz -90 deg; joints [34.363, -72.386, 110.458, -131.325, 48.714, 143.965]
  MoveL 890 to (177.4, 55.53, -113.42) mm, rotated rx -179.9 ry 0 rz -90 deg; joints [33.241, -73.443, 111.884, -132.783, 48.307, 145.118]
  MoveC 891 to (173.18, 55.53, -114.69) mm, rotated rx -179.9 ry 0 rz -90 deg; joints [33.058, -73.517, 111.986, -133.002, 48.221, 145.276] to (170.38, 55.53, -118.1) mm, rotated rx -179.9 ry 0 rz -90 deg; joints [32.876, -73.435, 111.881, -133.188, 48.102, 145.385]
  MoveL 892 to (170.38, 55.52, -118.1) mm, rotated rx -179.9 ry 0 rz -90 deg; joints [32.876, -73.435, 111.881, -133.188, 48.102, 145.385]
  MoveC 893 to (167.58, 55.53, -121.5) mm, rotated rx -179.9 ry 0 rz -90 deg; joints [32.695, -73.352, 111.776, -133.373, 47.983, 145.494] to (163.36, 55.52, -122.78) mm, rotated rx -179.9 ry 0 rz -90 deg; joints [32.512, -73.424, 111.874, -133.594, 47.897, 145.653]
  MoveL 894 to (163.36, 55.52, -122.78) mm, rotated rx -179.9 ry 0 rz -90 deg; joints [32.512, -73.424, 111.874, -133.594, 47.897, 145.653]
  MoveL 895 to (-199.47, 55.52, -122.78) mm, rotated rx -179.9 ry 0 rz -90 deg; joints [17.368, -82.92, 123.76, -153.997, 42.895, 160.839]
  MoveC 896 to (-202.2, 55.53, -123.91) mm, rotated rx -179.9 ry 0 rz -90 deg; joints [17.224, -82.903, 123.742, -154.197, 42.847, 160.983] to (-203.33, 55.53, -126.63) mm, rotated rx -179.9 ry 0 rz -90 deg; joints [17.132, -82.758, 123.579, -154.317, 42.801, 161.064]
  MoveL 897 to (-203.33, 55.53, -126.63) mm, rotated rx -179.9 ry 0 rz -90 deg; joints [17.132, -82.758, 123.579, -154.317, 42.801, 161.064]
  MoveL 898 to (-203.33, 55.53, -185.6) mm, rotated rx -179.9 ry 0 rz -90 deg; joints [16.318, -79.199, 119.436, -155.186, 42.008, 161.524]
  MoveC 899 to (-202.2, 55.53, -188.33) mm, rotated rx -179.9 ry 0 rz -90 deg; joints [16.332, -79.016, 119.216, -155.147, 41.979, 161.486] to (-199.47, 55.53, -189.46) mm, rotated rx -179.9 ry 0 rz -90 deg; joints [16.439, -78.902, 119.076, -154.985, 41.99, 161.359]
  MoveL 900 to (-199.47, 55.53, -189.46) mm, rotated rx -179.9 ry 0 rz -90 deg; joints [16.439, -78.902, 119.076, -154.985, 41.99, 161.359]
  MoveL 901 to (199.47, 55.52, -189.46) mm, rotated rx -179.9 ry 0 rz -90 deg; joints [32.286, -68.821, 105.631, -132.739, 46.645, 144.19]
  MoveC 902 to (202.2, 55.52, -188.33) mm, rotated rx -179.9 ry 0 rz -90 deg; joints [32.405, -68.791, 105.586, -132.596, 46.705, 144.086] to (203.33, 55.52, -185.6) mm, rotated rx -179.9 ry 0 rz -90 deg; joints [32.504, -68.895, 105.729, -132.514, 46.789, 144.052]
  MoveL 903 to (203.33, 55.52, -185.6) mm, rotated rx -179.9 ry 0 rz -90 deg; joints [32.504, -68.895, 105.729, -132.514, 46.789, 144.052]
  MoveL 904 to (203.33, 55.52, -126.63) mm, rotated rx -179.9 ry 0 rz -90 deg; joints [33.852, -71.904, 109.824, -131.774, 48.312, 144.169]
  MoveC 905 to (202.2, 55.52, -123.91) mm, rotated rx -179.9 ry 0 rz -90 deg; joints [33.877, -72.08, 110.06, -131.787, 48.367, 144.211] to (199.47, 55.53, -122.78) mm, rotated rx -179.9 ry 0 rz -90 deg; joints [33.808, -72.229, 110.261, -131.896, 48.361, 144.312]
  MoveL 906 to (199.47, 55.53, -122.78) mm, rotated rx -179.9 ry 0 rz -90 deg; joints [33.808, -72.229, 110.261, -131.896, 48.361, 144.312]
  MoveL 907 to (163.36, 55.52, -122.78) mm, rotated rx -179.9 ry 0 rz -90 deg; joints [32.512, -73.424, 111.874, -133.594, 47.897, 145.653]
  MoveC 908 to (159.14, 55.53, -124.06) mm, rotated rx -179.9 ry 0 rz -90 deg; joints [32.328, -73.495, 111.971, -133.815, 47.811, 145.813] to (156.34, 55.53, -127.46) mm, rotated rx -179.9 ry 0 rz -90 deg; joints [32.147, -73.409, 111.863, -134.002, 47.693, 145.923]
  MoveL 909 to (156.34, 55.52, -127.46) mm, rotated rx -179.9 ry 0 rz -90 deg; joints [32.147, -73.409, 111.863, -134.002, 47.693, 145.923]
  MoveC 910 to (153.54, 55.52, -130.86) mm, rotated rx -179.9 ry 0 rz -90 deg; joints [31.966, -73.323, 111.753, -134.189, 47.575, 146.033] to (149.32, 55.53, -132.14) mm, rotated rx -179.9 ry 0 rz -90 deg; joints [31.782, -73.391, 111.847, -134.412, 47.49, 146.195]
  MoveL 911 to (149.32, 55.52, -132.14) mm, rotated rx -179.9 ry 0 rz -90 deg; joints [31.782, -73.391, 111.847, -134.412, 47.49, 146.195]
  MoveL 912 to (-190.11, 55.52, -132.14) mm, rotated rx -179.9 ry 0 rz -90 deg; joints [17.665, -82.174, 122.908, -153.536, 42.899, 160.475]
  MoveC 913 to (-192.84, 55.52, -133.27) mm, rotated rx -179.9 ry 0 rz -90 deg; joints [17.522, -82.158, 122.891, -153.733, 42.851, 160.616] to (-193.96, 55.53, -135.99) mm, rotated rx -179.9 ry 0 rz -90 deg; joints [17.43, -82.014, 122.728, -153.851, 42.803, 160.696]
  MoveL 914 to (-193.96, 55.53, -135.99) mm, rotated rx -179.9 ry 0 rz -90 deg; joints [17.43, -82.014, 122.728, -153.851, 42.803, 160.696]
  MoveL 915 to (-193.96, 55.52, -176.24) mm, rotated rx -179.9 ry 0 rz -90 deg; joints [16.862, -79.594, 119.902, -154.451, 42.249, 161.009]
  MoveC 916 to (-192.84, 55.53, -178.97) mm, rotated rx -179.9 ry 0 rz -90 deg; joints [16.876, -79.411, 119.682, -154.415, 42.221, 160.972] to (-190.11, 55.52, -180.09) mm, rotated rx -179.9 ry 0 rz -90 deg; joints [16.982, -79.294, 119.541, -154.254, 42.234, 160.847]
  MoveL 917 to (-190.11, 55.53, -180.09) mm, rotated rx -179.9 ry 0 rz -90 deg; joints [16.982, -79.294, 119.541, -154.254, 42.234, 160.847]
  MoveL 918 to (190.11, 55.52, -180.09) mm, rotated rx -179.9 ry 0 rz -90 deg; joints [32.167, -69.606, 106.725, -133.085, 46.785, 144.591]
  MoveC 919 to (192.84, 55.52, -178.97) mm, rotated rx -179.9 ry 0 rz -90 deg; joints [32.287, -69.576, 106.681, -132.942, 46.846, 144.487] to (193.96, 55.52, -176.24) mm, rotated rx -179.9 ry 0 rz -90 deg; joints [32.387, -69.68, 106.823, -132.857, 46.93, 144.451]
  MoveL 920 to (193.96, 55.52, -176.24) mm, rotated rx -179.9 ry 0 rz -90 deg; joints [32.387, -69.68, 106.823, -132.857, 46.93, 144.451]
  MoveL 921 to (193.96, 55.53, -135.99) mm, rotated rx -179.9 ry 0 rz -90 deg; joints [33.302, -71.741, 109.617, -132.343, 47.96, 144.516]
  MoveC 922 to (192.84, 55.52, -133.27) mm, rotated rx -179.9 ry 0 rz -90 deg; joints [33.326, -71.918, 109.854, -132.358, 48.015, 144.559] to (190.11, 55.52, -132.14) mm, rotated rx -179.9 ry 0 rz -90 deg; joints [33.255, -72.065, 110.054, -132.469, 48.009, 144.661]
  MoveL 923 to (190.11, 55.53, -132.14) mm, rotated rx -179.9 ry 0 rz -90 deg; joints [33.255, -72.065, 110.054, -132.469, 48.009, 144.661]
  MoveL 924 to (149.32, 55.52, -132.14) mm, rotated rx -179.9 ry 0 rz -90 deg; joints [31.782, -73.391, 111.847, -134.412, 47.49, 146.195]
  MoveC 925 to (145.1, 55.53, -133.42) mm, rotated rx -179.9 ry 0 rz -90 deg; joints [31.598, -73.459, 111.94, -134.636, 47.405, 146.356] to (142.29, 55.52, -136.82) mm, rotated rx -179.9 ry 0 rz -90 deg; joints [31.417, -73.37, 111.827, -134.824, 47.287, 146.468]
  MoveL 926 to (142.29, 55.52, -136.82) mm, rotated rx -179.9 ry 0 rz -90 deg; joints [31.417, -73.37, 111.827, -134.824, 47.287, 146.468]
  MoveC 927 to (139.49, 55.53, -140.23) mm, rotated rx -179.9 ry 0 rz -90 deg; joints [31.237, -73.28, 111.712, -135.012, 47.17, 146.58] to (135.27, 55.52, -141.5) mm, rotated rx -179.9 ry 0 rz -90 deg; joints [31.053, -73.346, 111.802, -135.238, 47.086, 146.743]
  MoveL 928 to (135.27, 55.53, -141.5) mm, rotated rx -179.9 ry 0 rz -90 deg; joints [31.053, -73.346, 111.802, -135.238, 47.086, 146.743]
  MoveL 929 to (-180.75, 55.53, -141.5) mm, rotated rx -179.9 ry 0 rz -90 deg; joints [17.956, -81.43, 122.048, -153.078, 42.895, 160.108]
  MoveC 930 to (-183.47, 55.52, -142.63) mm, rotated rx -179.9 ry 0 rz -90 deg; joints [17.814, -81.415, 122.032, -153.273, 42.846, 160.248] to (-184.6, 55.52, -145.36) mm, rotated rx -179.9 ry 0 rz -90 deg; joints [17.723, -81.273, 121.868, -153.389, 42.795, 160.325]
  MoveL 931 to (-184.6, 55.53, -145.36) mm, rotated rx -179.9 ry 0 rz -90 deg; joints [17.723, -81.273, 121.868, -153.389, 42.795, 160.325]
  MoveL 932 to (-184.6, 55.52, -166.88) mm, rotated rx -179.9 ry 0 rz -90 deg; joints [17.413, -79.983, 120.357, -153.713, 42.493, 160.492]
  MoveC 933 to (-183.47, 55.52, -169.6) mm, rotated rx -179.9 ry 0 rz -90 deg; joints [17.425, -79.799, 120.139, -153.679, 42.465, 160.457] to (-180.75, 55.53, -170.73) mm, rotated rx -179.9 ry 0 rz -90 deg; joints [17.531, -79.681, 119.997, -153.52, 42.48, 160.334]
  MoveL 934 to (-180.75, 55.53, -170.73) mm, rotated rx -179.9 ry 0 rz -90 deg; joints [17.531, -79.681, 119.997, -153.52, 42.48, 160.334]
  MoveL 935 to (180.75, 55.52, -170.73) mm, rotated rx -179.9 ry 0 rz -90 deg; joints [32.045, -70.389, 107.807, -133.425, 46.92, 144.98]
  MoveC 936 to (183.47, 55.52, -169.6) mm, rotated rx -179.9 ry 0 rz -90 deg; joints [32.166, -70.36, 107.765, -133.281, 46.98, 144.876] to (184.6, 55.52, -166.88) mm, rotated rx -179.9 ry 0 rz -90 deg; joints [32.267, -70.464, 107.905, -133.193, 47.063, 144.837]
  MoveL 937 to (184.6, 55.53, -166.88) mm, rotated rx -179.9 ry 0 rz -90 deg; joints [32.267, -70.464, 107.905, -133.193, 47.063, 144.837]
  MoveL 938 to (184.6, 55.53, -145.36) mm, rotated rx -179.9 ry 0 rz -90 deg; joints [32.754, -71.571, 109.399, -132.914, 47.609, 144.864]
  MoveC 939 to (183.47, 55.52, -142.63) mm, rotated rx -179.9 ry 0 rz -90 deg; joints [32.776, -71.747, 109.636, -132.93, 47.664, 144.908] to (180.75, 55.52, -141.5) mm, rotated rx -179.9 ry 0 rz -90 deg; joints [32.705, -71.894, 109.836, -133.044, 47.659, 145.012]
  MoveL 940 to (180.75, 55.52, -141.5) mm, rotated rx -179.9 ry 0 rz -90 deg; joints [32.705, -71.894, 109.836, -133.044, 47.659, 145.012]
  MoveL 941 to (135.27, 55.53, -141.5) mm, rotated rx -179.9 ry 0 rz -90 deg; joints [31.053, -73.346, 111.802, -135.238, 47.086, 146.743]
  MoveC 942 to (131.05, 55.53, -142.78) mm, rotated rx -179.9 ry 0 rz -90 deg; joints [30.868, -73.41, 111.891, -135.464, 47.001, 146.907] to (128.25, 55.53, -146.18) mm, rotated rx -179.9 ry 0 rz -90 deg; joints [30.689, -73.318, 111.773, -135.653, 46.885, 147.02]
  MoveL 943 to (128.25, 55.53, -146.18) mm, rotated rx -179.9 ry 0 rz -90 deg; joints [30.689, -73.318, 111.773, -135.653, 46.885, 147.02]
  MoveC 944 to (125.45, 55.53, -149.59) mm, rotated rx -179.9 ry 0 rz -90 deg; joints [30.51, -73.225, 111.655, -135.842, 46.768, 147.133] to (121.23, 55.52, -150.87) mm, rotated rx -179.9 ry 0 rz -90 deg; joints [30.325, -73.287, 111.74, -136.07, 46.684, 147.298]
  MoveL 945 to (121.23, 55.53, -150.87) mm, rotated rx -179.9 ry 0 rz -90 deg; joints [30.325, -73.287, 111.74, -136.07, 46.684, 147.298]
  MoveL 946 to (-171.39, 55.52, -150.87) mm, rotated rx -179.9 ry 0 rz -90 deg; joints [18.241, -80.688, 121.178, -152.623, 42.88, 159.739]
  MoveC 947 to (-174.11, 55.53, -151.99) mm, rotated rx -179.9 ry 0 rz -90 deg; joints [18.101, -80.674, 121.163, -152.815, 42.831, 159.878] to (-175.24, 55.53, -154.72) mm, rotated rx -179.9 ry 0 rz -90 deg; joints [18.01, -80.533, 120.999, -152.929, 42.779, 159.953]
  MoveL 948 to (-175.24, 55.52, -154.72) mm, rotated rx -179.9 ry 0 rz -90 deg; joints [18.01, -80.533, 120.999, -152.929, 42.779, 159.953]
  MoveL 949 to (-175.24, 55.52, -157.52) mm, rotated rx -179.9 ry 0 rz -90 deg; joints [17.969, -80.365, 120.802, -152.972, 42.738, 159.975]
  MoveC 950 to (-174.11, 55.53, -160.24) mm, rotated rx -179.9 ry 0 rz -90 deg; joints [17.98, -80.181, 120.585, -152.94, 42.712, 159.941] to (-171.39, 55.52, -161.37) mm, rotated rx -179.9 ry 0 rz -90 deg; joints [18.085, -80.062, 120.442, -152.783, 42.728, 159.82]
  MoveL 951 to (-171.39, 55.52, -161.37) mm, rotated rx -179.9 ry 0 rz -90 deg; joints [18.085, -80.062, 120.442, -152.783, 42.728, 159.82]
  MoveL 952 to (171.39, 55.53, -161.37) mm, rotated rx -179.9 ry 0 rz -90 deg; joints [31.921, -71.173, 108.878, -133.758, 47.047, 145.357]
  MoveC 953 to (174.11, 55.53, -160.24) mm, rotated rx -179.9 ry 0 rz -90 deg; joints [32.044, -71.144, 108.836, -133.613, 47.108, 145.253] to (175.24, 55.52, -157.52) mm, rotated rx -179.9 ry 0 rz -90 deg; joints [32.145, -71.248, 108.976, -133.523, 47.19, 145.213]
  MoveL 954 to (175.24, 55.53, -157.52) mm, rotated rx -179.9 ry 0 rz -90 deg; joints [32.145, -71.248, 108.976, -133.523, 47.19, 145.213]
  MoveL 955 to (175.24, 55.52, -154.72) mm, rotated rx -179.9 ry 0 rz -90 deg; joints [32.208, -71.393, 109.17, -133.486, 47.26, 145.215]
  MoveC 956 to (174.11, 55.53, -151.99) mm, rotated rx -179.9 ry 0 rz -90 deg; joints [32.229, -71.57, 109.409, -133.504, 47.315, 145.26] to (171.39, 55.52, -150.87) mm, rotated rx -179.9 ry 0 rz -90 deg; joints [32.157, -71.715, 109.607, -133.619, 47.31, 145.365]
  MoveL 957 to (171.39, 55.52, -150.87) mm, rotated rx -179.9 ry 0 rz -90 deg; joints [32.157, -71.715, 109.607, -133.619, 47.31, 145.365]
  MoveL 958 to (121.23, 55.53, -150.87) mm, rotated rx -179.9 ry 0 rz -90 deg; joints [30.325, -73.287, 111.74, -136.07, 46.684, 147.298]
  MoveL 959 to (121.01, 55.54, -150.88) mm, rotated rx -179.9 ry 0 rz -90 deg; joints [30.316, -73.294, 111.747, -136.08, 46.68, 147.306]
  MoveL 960 to (120.8, 55.6, -150.94) mm, rotated rx -179.9 ry 0 rz -90 deg; joints [30.307, -73.299, 111.75, -136.089, 46.674, 147.31]
  MoveL 961 to (120.62, 55.7, -151.02) mm, rotated rx -179.9 ry 0 rz -90 deg; joints [30.299, -73.303, 111.748, -136.095, 46.665, 147.311]
  MoveL 962 to (120.47, 55.82, -151.12) mm, rotated rx -179.9 ry 0 rz -90 deg; joints [30.291, -73.307, 111.743, -136.099, 46.654, 147.309]
  MoveL 963 to (120.35, 55.98, -151.22) mm, rotated rx -179.9 ry 0 rz -90 deg; joints [30.284, -73.31, 111.736, -136.099, 46.643, 147.304]
  MoveL 964 to (120.26, 56.16, -151.31) mm, rotated rx -179.9 ry 0 rz -90 deg; joints [30.279, -73.313, 111.726, -136.097, 46.631, 147.296]
  MoveL 965 to (120.2, 56.36, -151.39) mm, rotated rx -179.9 ry 0 rz -90 deg; joints [30.275, -73.318, 111.717, -136.092, 46.618, 147.285]
  MoveL 966 to (120.17, 56.57, -151.43) mm, rotated rx -179.9 ry 0 rz -90 deg; joints [30.273, -73.323, 111.707, -136.085, 46.606, 147.273]
  MoveL 967 to (120.16, 56.8, -151.45) mm, rotated rx -179.9 ry 0 rz -90 deg; joints [30.272, -73.33, 111.699, -136.076, 46.595, 147.259]
  Set speed (1000.0 mm/s)
  MoveL 968 to (120.16, 110.53, -151.45) mm, rotated rx -179.9 ry 0 rz -90 deg; joints [30.245, -74.935, 109.673, -133.558, 44.02, 143.657]
  MoveL 969 to (319.15, 110.52, -150.09) mm, rotated rx -179.9 ry 0 rz -90 deg; joints [37.136, -68.142, 100.43, -124.321, 46.956, 135.924]
  MoveL 970 to (319.15, 83.04, -150.09) mm, rotated rx -179.9 ry 0 rz -90 deg; joints [37.15, -67.432, 101.479, -125.63, 47.973, 137.87]
  Set speed (100.0 mm/s)
  MoveL 971 to (319.13, 82.83, -150.09) mm, rotated rx -179.9 ry 0 rz -90 deg; joints [37.15, -67.427, 101.488, -125.64, 47.981, 137.886]
  MoveL 972 to (319.08, 82.62, -150.09) mm, rotated rx -179.9 ry 0 rz -90 deg; joints [37.148, -67.424, 101.499, -125.652, 47.989, 137.902]
  MoveL 973 to (318.99, 82.42, -150.09) mm, rotated rx -179.9 ry 0 rz -90 deg; joints [37.145, -67.422, 101.511, -125.665, 47.995, 137.919]
  MoveL 974 to (318.86, 82.24, -150.09) mm, rotated rx -179.9 ry 0 rz -90 deg; joints [37.141, -67.421, 101.523, -125.679, 48, 137.937]
  MoveL 975 to (318.71, 82.09, -150.1) mm, rotated rx -179.9 ry 0 rz -90 deg; joints [37.136, -67.422, 101.537, -125.693, 48.004, 137.953]
  MoveL 976 to (318.54, 81.96, -150.11) mm, rotated rx -179.9 ry 0 rz -90 deg; joints [37.131, -67.425, 101.55, -125.706, 48.006, 137.969]
  MoveL 977 to (318.35, 81.86, -150.13) mm, rotated rx -179.9 ry 0 rz -90 deg; joints [37.124, -67.428, 101.562, -125.719, 48.007, 137.983]
  MoveL 978 to (318.14, 81.8, -150.16) mm, rotated rx -179.9 ry 0 rz -90 deg; joints [37.117, -67.433, 101.574, -125.731, 48.006, 137.995]
  MoveL 979 to (317.93, 81.78, -150.19) mm, rotated rx -179.9 ry 0 rz -90 deg; joints [37.109, -67.438, 101.583, -125.742, 48.004, 138.004]
  MoveL 980 to (315.89, 81.7, -150.99) mm, rotated rx -179.9 ry 0 rz -90 deg; joints [37.026, -67.472, 101.639, -125.842, 47.96, 138.083]
  MoveL 981 to (314.27, 81.62, -152.45) mm, rotated rx -179.9 ry 0 rz -90 deg; joints [36.939, -67.458, 101.626, -125.93, 47.903, 138.141]
  MoveL 982 to (313.28, 81.54, -154.4) mm, rotated rx -179.9 ry 0 rz -90 deg; joints [36.86, -67.395, 101.546, -125.995, 47.84, 138.173]
  MoveL 983 to (313.05, 81.47, -156.57) mm, rotated rx -179.9 ry 0 rz -90 deg; joints [36.801, -67.294, 101.409, -126.029, 47.78, 138.173]
  MoveL 984 to (313.61, 81.39, -158.69) mm, rotated rx -179.9 ry 0 rz -90 deg; joints [36.768, -67.166, 101.235, -126.027, 47.73, 138.144]
  MoveL 985 to (314.88, 81.31, -160.46) mm, rotated rx -179.9 ry 0 rz -90 deg; joints [36.767, -67.029, 101.046, -125.99, 47.698, 138.088]
  MoveL 986 to (316.71, 81.24, -161.67) mm, rotated rx -179.9 ry 0 rz -90 deg; joints [36.796, -66.9, 100.867, -125.924, 47.689, 138.014]
  MoveL 987 to (318.84, 81.16, -162.15) mm, rotated rx -179.9 ry 0 rz -90 deg; joints [36.852, -66.796, 100.722, -125.839, 47.703, 137.933]
  MoveL 988 to (321, 81.08, -161.83) mm, rotated rx -179.9 ry 0 rz -90 deg; joints [36.928, -66.729, 100.631, -125.745, 47.74, 137.857]
  MoveL 989 to (322.91, 81.01, -160.77) mm, rotated rx -179.9 ry 0 rz -90 deg; joints [37.014, -66.709, 100.606, -125.656, 47.795, 137.795]
  MoveL 990 to (324.31, 80.93, -159.1) mm, rotated rx -179.9 ry 0 rz -90 deg; joints [37.098, -66.738, 100.651, -125.583, 47.861, 137.758]
  MoveL 991 to (325.03, 80.85, -157.03) mm, rotated rx -179.9 ry 0 rz -90 deg; joints [37.17, -66.811, 100.76, -125.538, 47.93, 137.75]
  MoveL 992 to (324.97, 80.78, -154.85) mm, rotated rx -179.9 ry 0 rz -90 deg; joints [37.221, -66.92, 100.919, -125.525, 47.994, 137.772]
  MoveL 993 to (324.13, 80.7, -152.83) mm, rotated rx -179.9 ry 0 rz -90 deg; joints [37.243, -67.049, 101.108, -125.547, 48.043, 137.824]
  MoveL 994 to (322.62, 80.62, -151.24) mm, rotated rx -179.9 ry 0 rz -90 deg; joints [37.233, -67.181, 101.302, -125.601, 48.073, 137.897]
  MoveL 995 to (320.65, 80.55, -150.3) mm, rotated rx -179.9 ry 0 rz -90 deg; joints [37.194, -67.299, 101.476, -125.681, 48.079, 137.984]
  MoveL 996 to (318.48, 80.47, -150.11) mm, rotated rx -179.9 ry 0 rz -90 deg; joints [37.129, -67.387, 101.608, -125.778, 48.061, 138.074]
  MoveL 997 to (316.38, 80.39, -150.72) mm, rotated rx -179.9 ry 0 rz -90 deg; joints [37.048, -67.433, 101.68, -125.878, 48.023, 138.156]
  MoveL 998 to (314.63, 80.32, -152.03) mm, rotated rx -179.9 ry 0 rz -90 deg; joints [36.961, -67.43, 101.685, -125.97, 47.968, 138.221]
  MoveL 999 to (313.47, 80.24, -153.88) mm, rotated rx -179.9 ry 0 rz -90 deg; joints [36.879, -67.38, 101.621, -126.042, 47.906, 138.259]
  MoveL 1000 to (313.04, 80.16, -156.02) mm, rotated rx -179.9 ry 0 rz -90 deg; joints [36.815, -67.287, 101.497, -126.084, 47.844, 138.268]
  MoveL 1001 to (313.4, 80.09, -158.18) mm, rotated rx -179.9 ry 0 rz -90 deg; joints [36.775, -67.165, 101.33, -126.092, 47.791, 138.245]
  MoveL 1002 to (314.5, 80.01, -160.06) mm, rotated rx -179.9 ry 0 rz -90 deg; joints [36.765, -67.028, 101.142, -126.064, 47.754, 138.196]
  MoveL 1003 to (316.21, 79.93, -161.43) mm, rotated rx -179.9 ry 0 rz -90 deg; joints [36.786, -66.896, 100.958, -126.005, 47.739, 138.125]
  MoveL 1004 to (318.29, 79.86, -162.1) mm, rotated rx -179.9 ry 0 rz -90 deg; joints [36.836, -66.783, 100.803, -125.923, 47.747, 138.045]
  MoveL 1005 to (320.47, 79.78, -161.99) mm, rotated rx -179.9 ry 0 rz -90 deg; joints [36.908, -66.706, 100.697, -125.83, 47.778, 137.967]
  MoveL 1006 to (322.47, 79.7, -161.1) mm, rotated rx -179.9 ry 0 rz -90 deg; joints [36.992, -66.674, 100.655, -125.738, 47.829, 137.9]
  MoveL 1007 to (324.02, 79.63, -159.56) mm, rotated rx -179.9 ry 0 rz -90 deg; joints [37.078, -66.691, 100.682, -125.661, 47.893, 137.856]
  MoveL 1008 to (324.92, 79.55, -157.57) mm, rotated rx -179.9 ry 0 rz -90 deg; joints [37.154, -66.754, 100.776, -125.607, 47.962, 137.84]
  MoveL 1009 to (325.06, 79.47, -155.39) mm, rotated rx -179.9 ry 0 rz -90 deg; joints [37.211, -66.854, 100.924, -125.586, 48.028, 137.856]
  MoveL 1010 to (324.41, 79.4, -153.31) mm, rotated rx -179.9 ry 0 rz -90 deg; joints [37.241, -66.98, 101.107, -125.599, 48.082, 137.9]
  MoveL 1011 to (323.06, 79.32, -151.59) mm, rotated rx -179.9 ry 0 rz -90 deg; joints [37.239, -67.113, 101.302, -125.645, 48.117, 137.969]
  MoveL 1012 to (321.18, 79.24, -150.47) mm, rotated rx -179.9 ry 0 rz -90 deg; joints [37.207, -67.236, 101.484, -125.72, 48.13, 138.053]
  MoveL 1013 to (319.03, 79.17, -150.09) mm, rotated rx -179.9 ry 0 rz -90 deg; joints [37.148, -67.332, 101.628, -125.813, 48.118, 138.143]
  MoveL 1014 to (316.88, 79.09, -150.49) mm, rotated rx -179.9 ry 0 rz -90 deg; joints [37.07, -67.39, 101.717, -125.914, 48.084, 138.228]
  MoveL 1015 to (315.02, 79.01, -151.64) mm, rotated rx -179.9 ry 0 rz -90 deg; joints [36.984, -67.4, 101.739, -126.01, 48.033, 138.298]
  MoveL 1016 to (313.7, 78.94, -153.37) mm, rotated rx -179.9 ry 0 rz -90 deg; joints [36.9, -67.361, 101.692, -126.088, 47.972, 138.344]
  MoveL 1017 to (313.07, 78.86, -155.47) mm, rotated rx -179.9 ry 0 rz -90 deg; joints [36.829, -67.278, 101.582, -126.138, 47.909, 138.36]
  MoveL 1018 to (313.23, 78.78, -157.65) mm, rotated rx -179.9 ry 0 rz -90 deg; joints [36.783, -67.162, 101.424, -126.154, 47.853, 138.345]
  MoveL 1019 to (314.16, 78.71, -159.63) mm, rotated rx -179.9 ry 0 rz -90 deg; joints [36.765, -67.027, 101.239, -126.135, 47.812, 138.302]
  MoveL 1020 to (315.73, 78.63, -161.14) mm, rotated rx -179.9 ry 0 rz -90 deg; joints [36.779, -66.892, 101.051, -126.083, 47.79, 138.236]
  MoveL 1021 to (317.74, 78.55, -162) mm, rotated rx -179.9 ry 0 rz -90 deg; joints [36.822, -66.773, 100.887, -126.006, 47.792, 138.157]
  MoveL 1022 to (319.92, 78.48, -162.09) mm, rotated rx -179.9 ry 0 rz -90 deg; joints [36.889, -66.687, 100.767, -125.915, 47.818, 138.077]
  MoveL 1023 to (322, 78.4, -161.39) mm, rotated rx -179.9 ry 0 rz -90 deg; joints [36.971, -66.642, 100.707, -125.821, 47.864, 138.007]
  MoveL 1024 to (323.68, 78.32, -160) mm, rotated rx -179.9 ry 0 rz -90 deg; joints [37.058, -66.647, 100.717, -125.739, 47.925, 137.956]
  MoveL 1025 to (324.76, 78.25, -158.11) mm, rotated rx -179.9 ry 0 rz -90 deg; joints [37.137, -66.698, 100.795, -125.679, 47.994, 137.933]
  MoveL 1026 to (325.1, 78.17, -155.95) mm, rotated rx -179.9 ry 0 rz -90 deg; joints [37.2, -66.791, 100.931, -125.649, 48.062, 137.94]
  MoveL 1027 to (324.64, 78.09, -153.81) mm, rotated rx -179.9 ry 0 rz -90 deg; joints [37.237, -66.911, 101.108, -125.653, 48.119, 137.978]
  MoveL 1028 to (323.45, 78.02, -151.98) mm, rotated rx -179.9 ry 0 rz -90 deg; joints [37.243, -67.044, 101.302, -125.691, 48.16, 138.041]
  MoveL 1029 to (321.69, 77.94, -150.69) mm, rotated rx -179.9 ry 0 rz -90 deg; joints [37.219, -67.171, 101.489, -125.76, 48.178, 138.122]
  MoveL 1030 to (319.58, 77.86, -150.11) mm, rotated rx -179.9 ry 0 rz -90 deg; joints [37.166, -67.275, 101.645, -125.849, 48.173, 138.212]
  MoveL 1031 to (317.41, 77.79, -150.32) mm, rotated rx -179.9 ry 0 rz -90 deg; joints [37.092, -67.344, 101.749, -125.949, 48.145, 138.299]
  MoveL 1032 to (315.45, 77.71, -151.29) mm, rotated rx -179.9 ry 0 rz -90 deg; joints [37.006, -67.366, 101.789, -126.047, 48.097, 138.374]
  MoveL 1033 to (313.97, 77.63, -152.89) mm, rotated rx -179.9 ry 0 rz -90 deg; joints [36.921, -67.339, 101.759, -126.131, 48.038, 138.426]
  MoveL 1034 to (313.16, 77.56, -154.92) mm, rotated rx -179.9 ry 0 rz -90 deg; joints [36.846, -67.267, 101.663, -126.189, 47.975, 138.45]
  MoveL 1035 to (313.12, 77.48, -157.11) mm, rotated rx -179.9 ry 0 rz -90 deg; joints [36.793, -67.158, 101.515, -126.215, 47.917, 138.443]
  MoveL 1036 to (313.86, 77.4, -159.16) mm, rotated rx -179.9 ry 0 rz -90 deg; joints [36.767, -67.026, 101.335, -126.204, 47.871, 138.406]
  MoveL 1037 to (315.29, 77.33, -160.82) mm, rotated rx -179.9 ry 0 rz -90 deg; joints [36.773, -66.89, 101.146, -126.16, 47.844, 138.345]
  MoveL 1038 to (317.21, 77.25, -161.86) mm, rotated rx -179.9 ry 0 rz -90 deg; joints [36.809, -66.765, 100.973, -126.088, 47.839, 138.269]
  MoveL 1039 to (319.37, 77.17, -162.14) mm, rotated rx -179.9 ry 0 rz -90 deg; joints [36.871, -66.669, 100.84, -125.999, 47.859, 138.188]
  MoveL 1040 to (321.5, 77.09, -161.64) mm, rotated rx -179.9 ry 0 rz -90 deg; joints [36.95, -66.614, 100.765, -125.905, 47.9, 138.114]
  MoveL 1041 to (323.31, 77.02, -160.41) mm, rotated rx -179.9 ry 0 rz -90 deg; joints [37.037, -66.605, 100.757, -125.819, 47.958, 138.058]
  MoveL 1042 to (324.56, 76.94, -158.62) mm, rotated rx -179.9 ry 0 rz -90 deg; joints [37.119, -66.646, 100.818, -125.752, 48.026, 138.027]
  MoveL 1043 to (325.09, 76.86, -156.5) mm, rotated rx -179.9 ry 0 rz -90 deg; joints [37.187, -66.729, 100.94, -125.714, 48.095, 138.027]
  MoveL 1044 to (324.83, 76.79, -154.33) mm, rotated rx -179.9 ry 0 rz -90 deg; joints [37.231, -66.843, 101.109, -125.709, 48.156, 138.057]
  MoveL 1045 to (323.82, 76.71, -152.4) mm, rotated rx -179.9 ry 0 rz -90 deg; joints [37.245, -66.974, 101.301, -125.739, 48.201, 138.114]
  MoveL 1046 to (322.18, 76.63, -150.95) mm, rotated rx -179.9 ry 0 rz -90 deg; joints [37.229, -67.104, 101.493, -125.8, 48.226, 138.192]
  MoveL 1047 to (320.13, 76.56, -150.18) mm, rotated rx -179.9 ry 0 rz -90 deg; joints [37.182, -67.216, 101.658, -125.886, 48.226, 138.281]
  MoveL 1048 to (317.95, 76.48, -150.19) mm, rotated rx -179.9 ry 0 rz -90 deg; joints [37.113, -67.294, 101.777, -125.984, 48.204, 138.37]
  MoveL 1049 to (315.91, 76.4, -150.98) mm, rotated rx -179.9 ry 0 rz -90 deg; joints [37.029, -67.329, 101.834, -126.084, 48.161, 138.448]
  MoveL 1050 to (314.29, 76.33, -152.44) mm, rotated rx -179.9 ry 0 rz -90 deg; joints [36.942, -67.314, 101.821, -126.172, 48.104, 138.507]
  MoveL 1051 to (313.29, 76.25, -154.38) mm, rotated rx -179.9 ry 0 rz -90 deg; joints [36.864, -67.253, 101.741, -126.238, 48.041, 138.538]
  MoveL 1052 to (313.05, 76.17, -156.56) mm, rotated rx -179.9 ry 0 rz -90 deg; joints [36.804, -67.152, 101.605, -126.272, 47.981, 138.539]
  MoveL 1053 to (313.6, 76.1, -158.67) mm, rotated rx -179.9 ry 0 rz -90 deg; joints [36.771, -67.025, 101.431, -126.271, 47.931, 138.509]
  MoveL 1054 to (314.87, 76.02, -160.45) mm, rotated rx -179.9 ry 0 rz -90 deg; joints [36.769, -66.888, 101.241, -126.235, 47.899, 138.454]
  MoveL 1055 to (316.69, 75.94, -161.66) mm, rotated rx -179.9 ry 0 rz -90 deg; joints [36.798, -66.759, 101.062, -126.169, 47.888, 138.38]
  MoveL 1056 to (318.82, 75.87, -162.14) mm, rotated rx -179.9 ry 0 rz -90 deg; joints [36.854, -66.654, 100.917, -126.083, 47.902, 138.299]
  MoveL 1057 to (320.98, 75.79, -161.84) mm, rotated rx -179.9 ry 0 rz -90 deg; joints [36.93, -66.588, 100.826, -125.989, 47.938, 138.223]
  MoveL 1058 to (322.89, 75.71, -160.78) mm, rotated rx -179.9 ry 0 rz -90 deg; joints [37.016, -66.567, 100.8, -125.9, 47.992, 138.161]
  MoveL 1059 to (324.3, 75.64, -159.11) mm, rotated rx -179.9 ry 0 rz -90 deg; joints [37.1, -66.595, 100.844, -125.827, 48.058, 138.124]
  MoveL 1060 to (325.03, 75.56, -157.05) mm, rotated rx -179.9 ry 0 rz -90 deg; joints [37.172, -66.668, 100.953, -125.781, 48.127, 138.115]
  MoveL 1061 to (324.97, 75.48, -154.87) mm, rotated rx -179.9 ry 0 rz -90 deg; joints [37.223, -66.776, 101.111, -125.768, 48.191, 138.138]
  MoveL 1062 to (324.14, 75.41, -152.85) mm, rotated rx -179.9 ry 0 rz -90 deg; joints [37.245, -66.905, 101.3, -125.789, 48.241, 138.189]
  MoveL 1063 to (322.64, 75.33, -151.26) mm, rotated rx -179.9 ry 0 rz -90 deg; joints [37.236, -67.037, 101.494, -125.843, 48.271, 138.262]
  MoveL 1064 to (320.67, 75.25, -150.3) mm, rotated rx -179.9 ry 0 rz -90 deg; joints [37.197, -67.154, 101.668, -125.923, 48.278, 138.349]
  MoveL 1065 to (318.5, 75.18, -150.11) mm, rotated rx -179.9 ry 0 rz -90 deg; joints [37.133, -67.242, 101.801, -126.019, 48.262, 138.439]
  MoveL 1066 to (316.39, 75.1, -150.71) mm, rotated rx -179.9 ry 0 rz -90 deg; joints [37.052, -67.288, 101.874, -126.12, 48.223, 138.521]
  MoveL 1067 to (314.64, 75.02, -152.02) mm, rotated rx -179.9 ry 0 rz -90 deg; joints [36.964, -67.286, 101.879, -126.212, 48.17, 138.585]
  MoveL 1068 to (313.47, 74.95, -153.86) mm, rotated rx -179.9 ry 0 rz -90 deg; joints [36.883, -67.236, 101.815, -126.284, 48.108, 138.624]
  MoveL 1069 to (313.04, 74.87, -156) mm, rotated rx -179.9 ry 0 rz -90 deg; joints [36.818, -67.144, 101.692, -126.327, 48.046, 138.633]
  MoveL 1070 to (313.39, 74.79, -158.16) mm, rotated rx -179.9 ry 0 rz -90 deg; joints [36.777, -67.022, 101.525, -126.335, 47.993, 138.611]
  MoveL 1071 to (314.49, 74.72, -160.05) mm, rotated rx -179.9 ry 0 rz -90 deg; joints [36.767, -66.886, 101.337, -126.308, 47.955, 138.561]
  MoveL 1072 to (316.19, 74.64, -161.42) mm, rotated rx -179.9 ry 0 rz -90 deg; joints [36.789, -66.754, 101.153, -126.249, 47.939, 138.491]
  MoveL 1073 to (318.27, 74.56, -162.1) mm, rotated rx -179.9 ry 0 rz -90 deg; joints [36.839, -66.642, 100.998, -126.167, 47.946, 138.411]
  MoveL 1074 to (320.45, 74.49, -161.99) mm, rotated rx -179.9 ry 0 rz -90 deg; joints [36.91, -66.565, 100.891, -126.074, 47.977, 138.332]
  MoveL 1075 to (322.45, 74.41, -161.11) mm, rotated rx -179.9 ry 0 rz -90 deg; joints [36.994, -66.532, 100.848, -125.982, 48.027, 138.266]
  MoveL 1076 to (324.01, 74.33, -159.58) mm, rotated rx -179.9 ry 0 rz -90 deg; joints [37.08, -66.548, 100.875, -125.904, 48.09, 138.221]
  MoveL 1077 to (324.92, 74.26, -157.59) mm, rotated rx -179.9 ry 0 rz -90 deg; joints [37.156, -66.61, 100.968, -125.85, 48.16, 138.205]
  MoveL 1078 to (325.06, 74.18, -155.41) mm, rotated rx -179.9 ry 0 rz -90 deg; joints [37.213, -66.711, 101.116, -125.828, 48.225, 138.22]
  MoveL 1079 to (324.42, 74.1, -153.33) mm, rotated rx -179.9 ry 0 rz -90 deg; joints [37.243, -66.835, 101.299, -125.84, 48.28, 138.265]
  MoveL 1080 to (323.07, 74.03, -151.6) mm, rotated rx -179.9 ry 0 rz -90 deg; joints [37.242, -66.968, 101.494, -125.887, 48.316, 138.333]
  MoveL 1081 to (321.2, 73.95, -150.47) mm, rotated rx -179.9 ry 0 rz -90 deg; joints [37.21, -67.091, 101.676, -125.961, 48.329, 138.417]
  MoveL 1082 to (319.05, 73.87, -150.09) mm, rotated rx -179.9 ry 0 rz -90 deg; joints [37.152, -67.187, 101.821, -126.054, 48.318, 138.507]
  MoveL 1083 to (316.9, 73.8, -150.49) mm, rotated rx -179.9 ry 0 rz -90 deg; joints [37.074, -67.245, 101.91, -126.155, 48.285, 138.592]
  MoveL 1084 to (315.04, 73.72, -151.63) mm, rotated rx -179.9 ry 0 rz -90 deg; joints [36.987, -67.255, 101.933, -126.251, 48.235, 138.662]
  MoveL 1085 to (313.7, 73.64, -153.36) mm, rotated rx -179.9 ry 0 rz -90 deg; joints [36.903, -67.217, 101.886, -126.329, 48.174, 138.708]
  MoveL 1086 to (313.07, 73.57, -155.45) mm, rotated rx -179.9 ry 0 rz -90 deg; joints [36.833, -67.135, 101.776, -126.38, 48.111, 138.724]
  MoveL 1087 to (313.23, 73.49, -157.63) mm, rotated rx -179.9 ry 0 rz -90 deg; joints [36.786, -67.019, 101.618, -126.397, 48.055, 138.71]
  MoveL 1088 to (314.15, 73.41, -159.61) mm, rotated rx -179.9 ry 0 rz -90 deg; joints [36.768, -66.885, 101.433, -126.378, 48.013, 138.666]
  MoveL 1089 to (315.72, 73.34, -161.13) mm, rotated rx -179.9 ry 0 rz -90 deg; joints [36.781, -66.75, 101.246, -126.326, 47.991, 138.601]
  MoveL 1090 to (317.72, 73.26, -162) mm, rotated rx -179.9 ry 0 rz -90 deg; joints [36.824, -66.631, 101.081, -126.25, 47.992, 138.522]
  MoveL 1091 to (319.91, 73.18, -162.09) mm, rotated rx -179.9 ry 0 rz -90 deg; joints [36.891, -66.544, 100.96, -126.158, 48.017, 138.442]
  MoveL 1092 to (321.98, 73.11, -161.4) mm, rotated rx -179.9 ry 0 rz -90 deg; joints [36.973, -66.5, 100.901, -126.065, 48.062, 138.372]
  MoveL 1093 to (323.67, 73.03, -160.02) mm, rotated rx -179.9 ry 0 rz -90 deg; joints [37.06, -66.504, 100.91, -125.982, 48.123, 138.321]
  MoveL 1094 to (324.76, 72.95, -158.12) mm, rotated rx -179.9 ry 0 rz -90 deg; joints [37.139, -66.555, 100.987, -125.921, 48.192, 138.297]
  MoveL 1095 to (325.1, 72.88, -155.97) mm, rotated rx -179.9 ry 0 rz -90 deg; joints [37.202, -66.646, 101.122, -125.89, 48.259, 138.305]
  MoveL 1096 to (324.65, 72.8, -153.83) mm, rotated rx -179.9 ry 0 rz -90 deg; joints [37.239, -66.766, 101.299, -125.894, 48.317, 138.342]
  MoveL 1097 to (323.47, 72.72, -151.99) mm, rotated rx -179.9 ry 0 rz -90 deg; joints [37.246, -66.899, 101.493, -125.932, 48.358, 138.405]
  MoveL 1098 to (321.71, 72.65, -150.69) mm, rotated rx -179.9 ry 0 rz -90 deg; joints [37.222, -67.025, 101.681, -126, 48.378, 138.486]
  MoveL 1099 to (319.6, 72.57, -150.11) mm, rotated rx -179.9 ry 0 rz -90 deg; joints [37.169, -67.13, 101.837, -126.089, 48.373, 138.576]
  MoveL 1100 to (317.43, 72.49, -150.31) mm, rotated rx -179.9 ry 0 rz -90 deg; joints [37.095, -67.198, 101.941, -126.189, 48.345, 138.663]
  MoveL 1101 to (315.47, 72.42, -151.28) mm, rotated rx -179.9 ry 0 rz -90 deg; joints [37.01, -67.221, 101.981, -126.288, 48.299, 138.737]
  MoveL 1102 to (313.98, 72.34, -152.88) mm, rotated rx -179.9 ry 0 rz -90 deg; joints [36.924, -67.195, 101.952, -126.372, 48.24, 138.79]
  MoveL 1103 to (313.16, 72.26, -154.9) mm, rotated rx -179.9 ry 0 rz -90 deg; joints [36.849, -67.123, 101.857, -126.43, 48.177, 138.814]
  MoveL 1104 to (313.11, 72.18, -157.09) mm, rotated rx -179.9 ry 0 rz -90 deg; joints [36.796, -67.014, 101.71, -126.456, 48.119, 138.807]
  MoveL 1105 to (313.85, 72.11, -159.14) mm, rotated rx -179.9 ry 0 rz -90 deg; joints [36.77, -66.883, 101.529, -126.446, 48.072, 138.77]
  MoveL 1106 to (315.27, 72.03, -160.8) mm, rotated rx -179.9 ry 0 rz -90 deg; joints [36.776, -66.747, 101.34, -126.402, 48.045, 138.71]
  MoveL 1107 to (317.19, 71.95, -161.85) mm, rotated rx -179.9 ry 0 rz -90 deg; joints [36.812, -66.623, 101.167, -126.331, 48.04, 138.633]
  MoveL 1108 to (319.35, 71.88, -162.14) mm, rotated rx -179.9 ry 0 rz -90 deg; joints [36.873, -66.526, 101.034, -126.242, 48.059, 138.552]
  MoveL 1109 to (321.48, 71.8, -161.65) mm, rotated rx -179.9 ry 0 rz -90 deg; joints [36.952, -66.471, 100.957, -126.148, 48.099, 138.479]
  MoveL 1110 to (323.29, 71.72, -160.42) mm, rotated rx -179.9 ry 0 rz -90 deg; joints [37.039, -66.462, 100.949, -126.061, 48.157, 138.422]
  MoveL 1111 to (324.55, 71.65, -158.64) mm, rotated rx -179.9 ry 0 rz -90 deg; joints [37.121, -66.502, 101.009, -125.994, 48.224, 138.391]
  MoveL 1112 to (325.09, 71.57, -156.52) mm, rotated rx -179.9 ry 0 rz -90 deg; joints [37.189, -66.584, 101.131, -125.955, 48.293, 138.391]
  MoveL 1113 to (324.84, 71.49, -154.35) mm, rotated rx -179.9 ry 0 rz -90 deg; joints [37.233, -66.698, 101.3, -125.95, 48.354, 138.42]
  MoveL 1114 to (323.83, 71.42, -152.41) mm, rotated rx -179.9 ry 0 rz -90 deg; joints [37.248, -66.829, 101.492, -125.979, 48.4, 138.477]
  MoveL 1115 to (322.19, 71.34, -150.96) mm, rotated rx -179.9 ry 0 rz -90 deg; joints [37.232, -66.959, 101.683, -126.04, 48.425, 138.555]
  MoveL 1116 to (320.15, 71.26, -150.18) mm, rotated rx -179.9 ry 0 rz -90 deg; joints [37.186, -67.07, 101.849, -126.125, 48.427, 138.643]
  MoveL 1117 to (317.97, 71.19, -150.19) mm, rotated rx -179.9 ry 0 rz -90 deg; joints [37.116, -67.149, 101.969, -126.224, 48.405, 138.732]
  MoveL 1118 to (315.93, 71.11, -150.97) mm, rotated rx -179.9 ry 0 rz -90 deg; joints [37.032, -67.183, 102.026, -126.324, 48.363, 138.811]
  MoveL 1119 to (314.3, 71.03, -152.42) mm, rotated rx -179.9 ry 0 rz -90 deg; joints [36.946, -67.169, 102.014, -126.412, 48.306, 138.87]
  MoveL 1120 to (313.3, 70.96, -154.37) mm, rotated rx -179.9 ry 0 rz -90 deg; joints [36.867, -67.108, 101.934, -126.478, 48.244, 138.901]
  MoveL 1121 to (313.05, 70.88, -156.54) mm, rotated rx -179.9 ry 0 rz -90 deg; joints [36.807, -67.008, 101.799, -126.513, 48.183, 138.902]
  MoveL 1122 to (313.59, 70.8, -158.65) mm, rotated rx -179.9 ry 0 rz -90 deg; joints [36.774, -66.881, 101.624, -126.512, 48.133, 138.873]
  MoveL 1123 to (314.86, 70.73, -160.44) mm, rotated rx -179.9 ry 0 rz -90 deg; joints [36.772, -66.745, 101.435, -126.477, 48.1, 138.817]
  MoveL 1124 to (316.67, 70.65, -161.65) mm, rotated rx -179.9 ry 0 rz -90 deg; joints [36.8, -66.616, 101.256, -126.411, 48.089, 138.744]
  MoveL 1125 to (318.8, 70.57, -162.14) mm, rotated rx -179.9 ry 0 rz -90 deg; joints [36.856, -66.511, 101.11, -126.326, 48.102, 138.663]
  MoveL 1126 to (320.96, 70.5, -161.84) mm, rotated rx -179.9 ry 0 rz -90 deg; joints [36.932, -66.444, 101.018, -126.231, 48.137, 138.586]
  MoveL 1127 to (322.88, 70.42, -160.79) mm, rotated rx -179.9 ry 0 rz -90 deg; joints [37.018, -66.423, 100.992, -126.142, 48.191, 138.525]
  MoveL 1128 to (324.3, 70.34, -159.13) mm, rotated rx -179.9 ry 0 rz -90 deg; joints [37.102, -66.451, 101.036, -126.068, 48.256, 138.487]
  MoveL 1129 to (325.02, 70.27, -157.07) mm, rotated rx -179.9 ry 0 rz -90 deg; joints [37.174, -66.524, 101.143, -126.022, 48.325, 138.478]
  MoveL 1130 to (324.97, 70.19, -154.89) mm, rotated rx -179.9 ry 0 rz -90 deg; joints [37.225, -66.631, 101.302, -126.008, 48.389, 138.501]
  MoveL 1131 to (324.15, 70.11, -152.86) mm, rotated rx -179.9 ry 0 rz -90 deg; joints [37.248, -66.759, 101.49, -126.028, 48.44, 138.551]
  MoveL 1132 to (322.65, 70.04, -151.27) mm, rotated rx -179.9 ry 0 rz -90 deg; joints [37.239, -66.89, 101.684, -126.082, 48.471, 138.624]
  MoveL 1133 to (320.69, 69.96, -150.31) mm, rotated rx -179.9 ry 0 rz -90 deg; joints [37.2, -67.008, 101.859, -126.161, 48.479, 138.711]
  MoveL 1134 to (318.52, 69.88, -150.11) mm, rotated rx -179.9 ry 0 rz -90 deg; joints [37.136, -67.096, 101.992, -126.258, 48.463, 138.801]
  MoveL 1135 to (316.41, 69.81, -150.7) mm, rotated rx -179.9 ry 0 rz -90 deg; joints [37.055, -67.142, 102.065, -126.359, 48.425, 138.883]
  MoveL 1136 to (314.66, 69.73, -152) mm, rotated rx -179.9 ry 0 rz -90 deg; joints [36.968, -67.141, 102.071, -126.451, 48.372, 138.947]
  MoveL 1137 to (313.48, 69.65, -153.84) mm, rotated rx -179.9 ry 0 rz -90 deg; joints [36.886, -67.091, 102.008, -126.524, 48.31, 138.986]
  MoveL 1138 to (313.04, 69.58, -155.98) mm, rotated rx -179.9 ry 0 rz -90 deg; joints [36.821, -67, 101.885, -126.567, 48.248, 138.995]
  MoveL 1139 to (313.38, 69.5, -158.14) mm, rotated rx -179.9 ry 0 rz -90 deg; joints [36.78, -66.878, 101.718, -126.576, 48.195, 138.973]
  MoveL 1140 to (314.48, 69.42, -160.03) mm, rotated rx -179.9 ry 0 rz -90 deg; joints [36.77, -66.743, 101.53, -126.549, 48.157, 138.924]
  MoveL 1141 to (316.17, 69.35, -161.41) mm, rotated rx -179.9 ry 0 rz -90 deg; joints [36.791, -66.61, 101.346, -126.49, 48.14, 138.854]
  MoveL 1142 to (318.25, 69.27, -162.09) mm, rotated rx -179.9 ry 0 rz -90 deg; joints [36.841, -66.498, 101.19, -126.408, 48.147, 138.774]
  MoveL 1143 to (320.43, 69.19, -161.99) mm, rotated rx -179.9 ry 0 rz -90 deg; joints [36.912, -66.421, 101.083, -126.315, 48.176, 138.695]
  MoveL 1144 to (322.43, 69.12, -161.12) mm, rotated rx -179.9 ry 0 rz -90 deg; joints [36.996, -66.388, 101.04, -126.223, 48.226, 138.629]
  MoveL 1145 to (324, 69.04, -159.6) mm, rotated rx -179.9 ry 0 rz -90 deg; joints [37.082, -66.403, 101.066, -126.145, 48.289, 138.584]
  MoveL 1146 to (324.91, 68.96, -157.61) mm, rotated rx -179.9 ry 0 rz -90 deg; joints [37.159, -66.465, 101.158, -126.09, 48.358, 138.568]
  MoveL 1147 to (325.06, 68.89, -155.43) mm, rotated rx -179.9 ry 0 rz -90 deg; joints [37.216, -66.565, 101.306, -126.067, 48.424, 138.582]
  MoveL 1148 to (324.42, 68.81, -153.34) mm, rotated rx -179.9 ry 0 rz -90 deg; joints [37.246, -66.689, 101.489, -126.079, 48.479, 138.626]
  MoveL 1149 to (323.08, 68.73, -151.62) mm, rotated rx -179.9 ry 0 rz -90 deg; joints [37.245, -66.821, 101.684, -126.125, 48.515, 138.695]
  MoveL 1150 to (321.22, 68.66, -150.48) mm, rotated rx -179.9 ry 0 rz -90 deg; joints [37.213, -66.944, 101.865, -126.199, 48.529, 138.779]
  MoveL 1151 to (319.07, 68.58, -150.09) mm, rotated rx -179.9 ry 0 rz -90 deg; joints [37.155, -67.041, 102.011, -126.292, 48.519, 138.869]
  MoveL 1152 to (316.92, 68.5, -150.48) mm, rotated rx -179.9 ry 0 rz -90 deg; joints [37.077, -67.098, 102.101, -126.393, 48.487, 138.954]
  MoveL 1153 to (315.05, 68.43, -151.62) mm, rotated rx -179.9 ry 0 rz -90 deg; joints [36.99, -67.109, 102.124, -126.489, 48.437, 139.024]
  MoveL 1154 to (313.71, 68.35, -153.34) mm, rotated rx -179.9 ry 0 rz -90 deg; joints [36.906, -67.071, 102.077, -126.568, 48.377, 139.07]
  MoveL 1155 to (313.07, 68.27, -155.43) mm, rotated rx -179.9 ry 0 rz -90 deg; joints [36.836, -66.989, 101.968, -126.619, 48.314, 139.086]
  MoveL 1156 to (313.22, 68.2, -157.61) mm, rotated rx -179.9 ry 0 rz -90 deg; joints [36.789, -66.874, 101.811, -126.637, 48.258, 139.072]
  MoveL 1157 to (314.14, 68.12, -159.59) mm, rotated rx -179.9 ry 0 rz -90 deg; joints [36.77, -66.741, 101.626, -126.618, 48.215, 139.029]
  MoveL 1158 to (315.7, 68.04, -161.12) mm, rotated rx -179.9 ry 0 rz -90 deg; joints [36.784, -66.606, 101.438, -126.567, 48.193, 138.963]
  MoveL 1159 to (317.7, 67.97, -161.99) mm, rotated rx -179.9 ry 0 rz -90 deg; joints [36.826, -66.487, 101.273, -126.49, 48.193, 138.885]
  MoveL 1160 to (319.89, 67.89, -162.09) mm, rotated rx -179.9 ry 0 rz -90 deg; joints [36.893, -66.4, 101.152, -126.399, 48.217, 138.804]
  MoveL 1161 to (321.96, 67.81, -161.41) mm, rotated rx -179.9 ry 0 rz -90 deg; joints [36.975, -66.355, 101.092, -126.305, 48.262, 138.734]
  MoveL 1162 to (323.66, 67.73, -160.03) mm, rotated rx -179.9 ry 0 rz -90 deg; joints [37.062, -66.359, 101.1, -126.222, 48.322, 138.683]
  MoveL 1163 to (324.75, 67.66, -158.14) mm, rotated rx -179.9 ry 0 rz -90 deg; joints [37.141, -66.409, 101.177, -126.161, 48.39, 138.659]
  MoveL 1164 to (325.1, 67.58, -155.98) mm, rotated rx -179.9 ry 0 rz -90 deg; joints [37.204, -66.5, 101.312, -126.129, 48.458, 138.666]
  MoveL 1165 to (324.66, 67.5, -153.84) mm, rotated rx -179.9 ry 0 rz -90 deg; joints [37.242, -66.62, 101.488, -126.132, 48.516, 138.703]
  MoveL 1166 to (323.48, 67.43, -152) mm, rotated rx -179.9 ry 0 rz -90 deg; joints [37.249, -66.751, 101.682, -126.17, 48.558, 138.766]
  MoveL 1167 to (321.73, 67.35, -150.7) mm, rotated rx -179.9 ry 0 rz -90 deg; joints [37.225, -66.878, 101.87, -126.237, 48.578, 138.847]
  MoveL 1168 to (319.62, 67.27, -150.11) mm, rotated rx -179.9 ry 0 rz -90 deg; joints [37.173, -66.983, 102.026, -126.327, 48.574, 138.936]
  MoveL 1169 to (317.45, 67.2, -150.31) mm, rotated rx -179.9 ry 0 rz -90 deg; joints [37.099, -67.051, 102.131, -126.427, 48.547, 139.024]
  MoveL 1170 to (315.48, 67.12, -151.27) mm, rotated rx -179.9 ry 0 rz -90 deg; joints [37.013, -67.074, 102.172, -126.525, 48.502, 139.098]
  MoveL 1171 to (313.99, 67.04, -152.86) mm, rotated rx -179.9 ry 0 rz -90 deg; joints [36.927, -67.048, 102.143, -126.609, 48.443, 139.151]
  MoveL 1172 to (313.16, 66.97, -154.88) mm, rotated rx -179.9 ry 0 rz -90 deg; joints [36.852, -66.977, 102.049, -126.669, 48.38, 139.175]
  MoveL 1173 to (313.11, 66.89, -157.07) mm, rotated rx -179.9 ry 0 rz -90 deg; joints [36.799, -66.869, 101.901, -126.695, 48.322, 139.168]
  MoveL 1174 to (313.84, 66.81, -159.13) mm, rotated rx -179.9 ry 0 rz -90 deg; joints [36.773, -66.738, 101.721, -126.686, 48.275, 139.132]
  MoveL 1175 to (315.26, 66.74, -160.79) mm, rotated rx -179.9 ry 0 rz -90 deg; joints [36.778, -66.602, 101.532, -126.642, 48.247, 139.071]
  MoveL 1176 to (317.17, 66.66, -161.84) mm, rotated rx -179.9 ry 0 rz -90 deg; joints [36.814, -66.478, 101.359, -126.571, 48.241, 138.995]
  MoveL 1177 to (319.33, 66.58, -162.14) mm, rotated rx -179.9 ry 0 rz -90 deg; joints [36.875, -66.382, 101.225, -126.482, 48.259, 138.914]
  MoveL 1178 to (321.46, 66.51, -161.65) mm, rotated rx -179.9 ry 0 rz -90 deg; joints [36.954, -66.326, 101.148, -126.388, 48.299, 138.84]
  MoveL 1179 to (323.28, 66.43, -160.44) mm, rotated rx -179.9 ry 0 rz -90 deg; joints [37.041, -66.317, 101.139, -126.301, 48.356, 138.784]
  MoveL 1180 to (324.54, 66.35, -158.65) mm, rotated rx -179.9 ry 0 rz -90 deg; joints [37.123, -66.356, 101.199, -126.233, 48.423, 138.753]
  MoveL 1181 to (325.09, 66.28, -156.54) mm, rotated rx -179.9 ry 0 rz -90 deg; joints [37.191, -66.438, 101.32, -126.194, 48.491, 138.752]
  MoveL 1182 to (324.84, 66.2, -154.37) mm, rotated rx -179.9 ry 0 rz -90 deg; joints [37.236, -66.551, 101.488, -126.188, 48.553, 138.781]
  MoveL 1183 to (323.84, 66.12, -152.43) mm, rotated rx -179.9 ry 0 rz -90 deg; joints [37.251, -66.681, 101.68, -126.217, 48.599, 138.838]
  MoveL 1184 to (322.21, 66.05, -150.97) mm, rotated rx -179.9 ry 0 rz -90 deg; joints [37.234, -66.811, 101.872, -126.277, 48.625, 138.915]
  MoveL 1185 to (320.17, 65.97, -150.19) mm, rotated rx -179.9 ry 0 rz -90 deg; joints [37.189, -66.922, 102.038, -126.362, 48.628, 139.004]
  MoveL 1186 to (317.99, 65.89, -150.18) mm, rotated rx -179.9 ry 0 rz -90 deg; joints [37.12, -67.001, 102.158, -126.46, 48.607, 139.092]
  MoveL 1187 to (315.94, 65.82, -150.96) mm, rotated rx -179.9 ry 0 rz -90 deg; joints [37.036, -67.036, 102.215, -126.56, 48.565, 139.171]
  MoveL 1188 to (314.31, 65.74, -152.41) mm, rotated rx -179.9 ry 0 rz -90 deg; joints [36.949, -67.022, 102.204, -126.649, 48.509, 139.23]
  MoveL 1189 to (313.3, 65.66, -154.35) mm, rotated rx -179.9 ry 0 rz -90 deg; joints [36.87, -66.962, 102.125, -126.716, 48.447, 139.262]
  MoveL 1190 to (313.05, 65.59, -156.52) mm, rotated rx -179.9 ry 0 rz -90 deg; joints [36.81, -66.862, 101.99, -126.751, 48.386, 139.263]
  MoveL 1191 to (313.59, 65.51, -158.64) mm, rotated rx -179.9 ry 0 rz -90 deg; joints [36.777, -66.736, 101.816, -126.751, 48.336, 139.233]
  MoveL 1192 to (314.84, 65.43, -160.42) mm, rotated rx -179.9 ry 0 rz -90 deg; joints [36.774, -66.599, 101.626, -126.716, 48.302, 139.178]
  MoveL 1193 to (316.65, 65.36, -161.65) mm, rotated rx -179.9 ry 0 rz -90 deg; joints [36.803, -66.471, 101.447, -126.651, 48.291, 139.105]
  MoveL 1194 to (318.78, 65.28, -162.14) mm, rotated rx -179.9 ry 0 rz -90 deg; joints [36.858, -66.366, 101.301, -126.565, 48.303, 139.024]
  MoveL 1195 to (320.95, 65.2, -161.85) mm, rotated rx -179.9 ry 0 rz -90 deg; joints [36.934, -66.299, 101.208, -126.471, 48.337, 138.947]
  MoveL 1196 to (322.87, 65.13, -160.81) mm, rotated rx -179.9 ry 0 rz -90 deg; joints [37.019, -66.278, 101.182, -126.381, 48.39, 138.886]
  MoveL 1197 to (324.29, 65.05, -159.15) mm, rotated rx -179.9 ry 0 rz -90 deg; joints [37.104, -66.305, 101.224, -126.307, 48.456, 138.847]
  MoveL 1198 to (325.02, 64.97, -157.09) mm, rotated rx -179.9 ry 0 rz -90 deg; joints [37.177, -66.377, 101.332, -126.26, 48.525, 138.839]
  MoveL 1199 to (324.98, 64.9, -154.9) mm, rotated rx -179.9 ry 0 rz -90 deg; joints [37.228, -66.483, 101.49, -126.245, 48.589, 138.861]
  MoveL 1200 to (324.16, 64.82, -152.88) mm, rotated rx -179.9 ry 0 rz -90 deg; joints [37.251, -66.611, 101.678, -126.265, 48.64, 138.911]
  MoveL 1201 to (322.67, 64.74, -151.28) mm, rotated rx -179.9 ry 0 rz -90 deg; joints [37.242, -66.742, 101.872, -126.318, 48.671, 138.984]
  MoveL 1202 to (320.71, 64.67, -150.31) mm, rotated rx -179.9 ry 0 rz -90 deg; joints [37.203, -66.86, 102.047, -126.398, 48.68, 139.071]
  MoveL 1203 to (318.53, 64.59, -150.11) mm, rotated rx -179.9 ry 0 rz -90 deg; joints [37.139, -66.948, 102.18, -126.494, 48.664, 139.16]
  MoveL 1204 to (316.43, 64.51, -150.69) mm, rotated rx -179.9 ry 0 rz -90 deg; joints [37.058, -66.994, 102.254, -126.595, 48.628, 139.243]
  MoveL 1205 to (314.67, 64.44, -151.99) mm, rotated rx -179.9 ry 0 rz -90 deg; joints [36.971, -66.993, 102.261, -126.688, 48.575, 139.307]
  MoveL 1206 to (313.49, 64.36, -153.83) mm, rotated rx -179.9 ry 0 rz -90 deg; joints [36.89, -66.944, 102.198, -126.761, 48.514, 139.346]
  MoveL 1207 to (313.04, 64.28, -155.96) mm, rotated rx -179.9 ry 0 rz -90 deg; joints [36.824, -66.853, 102.075, -126.805, 48.452, 139.355]
  MoveL 1208 to (313.38, 64.21, -158.12) mm, rotated rx -179.9 ry 0 rz -90 deg; joints [36.783, -66.732, 101.909, -126.813, 48.398, 139.333]
  MoveL 1209 to (314.47, 64.13, -160.02) mm, rotated rx -179.9 ry 0 rz -90 deg; joints [36.773, -66.597, 101.721, -126.787, 48.36, 139.284]
  MoveL 1210 to (316.16, 64.05, -161.4) mm, rotated rx -179.9 ry 0 rz -90 deg; joints [36.793, -66.465, 101.537, -126.729, 48.342, 139.214]
  MoveL 1211 to (318.23, 63.98, -162.09) mm, rotated rx -179.9 ry 0 rz -90 deg; joints [36.843, -66.353, 101.38, -126.647, 48.348, 139.134]
  MoveL 1212 to (320.41, 63.9, -162) mm, rotated rx -179.9 ry 0 rz -90 deg; joints [36.914, -66.275, 101.273, -126.554, 48.377, 139.055]
  MoveL 1213 to (322.42, 63.82, -161.13) mm, rotated rx -179.9 ry 0 rz -90 deg; joints [36.998, -66.242, 101.229, -126.461, 48.426, 138.989]
  MoveL 1214 to (323.99, 63.75, -159.61) mm, rotated rx -179.9 ry 0 rz -90 deg; joints [37.084, -66.257, 101.254, -126.383, 48.489, 138.944]
  MoveL 1215 to (324.91, 63.67, -157.63) mm, rotated rx -179.9 ry 0 rz -90 deg; joints [37.161, -66.318, 101.346, -126.328, 48.557, 138.928]
  MoveL 1216 to (325.06, 63.59, -155.45) mm, rotated rx -179.9 ry 0 rz -90 deg; joints [37.218, -66.417, 101.493, -126.304, 48.623, 138.942]
  MoveL 1217 to (324.43, 63.52, -153.36) mm, rotated rx -179.9 ry 0 rz -90 deg; joints [37.248, -66.541, 101.676, -126.316, 48.678, 138.986]
  MoveL 1218 to (323.1, 63.44, -151.63) mm, rotated rx -179.9 ry 0 rz -90 deg; joints [37.248, -66.673, 101.871, -126.361, 48.716, 139.054]
  MoveL 1219 to (321.24, 63.36, -150.49) mm, rotated rx -179.9 ry 0 rz -90 deg; joints [37.217, -66.795, 102.053, -126.434, 48.73, 139.138]
  MoveL 1220 to (319.09, 63.29, -150.09) mm, rotated rx -179.9 ry 0 rz -90 deg; joints [37.158, -66.892, 102.198, -126.527, 48.721, 139.228]
  MoveL 1221 to (316.94, 63.21, -150.47) mm, rotated rx -179.9 ry 0 rz -90 deg; joints [37.081, -66.95, 102.289, -126.628, 48.69, 139.313]
  MoveL 1222 to (315.07, 63.13, -151.6) mm, rotated rx -179.9 ry 0 rz -90 deg; joints [36.994, -66.961, 102.313, -126.725, 48.64, 139.383]
  MoveL 1223 to (313.72, 63.05, -153.32) mm, rotated rx -179.9 ry 0 rz -90 deg; joints [36.91, -66.923, 102.267, -126.804, 48.58, 139.429]
  MoveL 1224 to (313.08, 62.98, -155.41) mm, rotated rx -179.9 ry 0 rz -90 deg; joints [36.839, -66.842, 102.158, -126.856, 48.518, 139.445]
  MoveL 1225 to (313.22, 62.9, -157.59) mm, rotated rx -179.9 ry 0 rz -90 deg; joints [36.791, -66.727, 102.001, -126.874, 48.461, 139.431]
  MoveL 1226 to (314.13, 62.82, -159.58) mm, rotated rx -179.9 ry 0 rz -90 deg; joints [36.773, -66.594, 101.816, -126.856, 48.418, 139.388]
  MoveL 1227 to (315.68, 62.75, -161.11) mm, rotated rx -179.9 ry 0 rz -90 deg; joints [36.786, -66.46, 101.629, -126.805, 48.395, 139.323]
  MoveL 1228 to (317.69, 62.67, -161.99) mm, rotated rx -179.9 ry 0 rz -90 deg; joints [36.829, -66.341, 101.463, -126.728, 48.395, 139.244]
  MoveL 1229 to (319.87, 62.59, -162.1) mm, rotated rx -179.9 ry 0 rz -90 deg; joints [36.895, -66.254, 101.341, -126.637, 48.418, 139.164]
  MoveL 1230 to (321.94, 62.52, -161.42) mm, rotated rx -179.9 ry 0 rz -90 deg; joints [36.977, -66.209, 101.28, -126.543, 48.462, 139.093]
  MoveL 1231 to (323.64, 62.44, -160.05) mm, rotated rx -179.9 ry 0 rz -90 deg; joints [37.064, -66.212, 101.288, -126.459, 48.522, 139.043]
  MoveL 1232 to (324.74, 62.36, -158.16) mm, rotated rx -179.9 ry 0 rz -90 deg; joints [37.143, -66.262, 101.364, -126.398, 48.59, 139.019]
  MoveL 1233 to (325.1, 62.29, -156) mm, rotated rx -179.9 ry 0 rz -90 deg; joints [37.206, -66.352, 101.499, -126.366, 48.658, 139.025]
  MoveL 1234 to (324.66, 62.21, -153.86) mm, rotated rx -179.9 ry 0 rz -90 deg; joints [37.244, -66.471, 101.675, -126.368, 48.716, 139.062]
  MoveL 1235 to (323.49, 62.13, -152.02) mm, rotated rx -179.9 ry 0 rz -90 deg; joints [37.252, -66.603, 101.869, -126.405, 48.758, 139.124]
  MoveL 1236 to (321.74, 62.06, -150.71) mm, rotated rx -179.9 ry 0 rz -90 deg; joints [37.228, -66.729, 102.056, -126.472, 48.779, 139.205]
  MoveL 1237 to (319.64, 61.98, -150.11) mm, rotated rx -179.9 ry 0 rz -90 deg; joints [37.176, -66.833, 102.213, -126.561, 48.776, 139.295]
  MoveL 1238 to (317.46, 61.9, -150.3) mm, rotated rx -179.9 ry 0 rz -90 deg; joints [37.102, -66.902, 102.319, -126.661, 48.75, 139.382]
  MoveL 1239 to (315.5, 61.83, -151.25) mm, rotated rx -179.9 ry 0 rz -90 deg; joints [37.017, -66.925, 102.36, -126.76, 48.705, 139.456]
  MoveL 1240 to (314, 61.75, -152.85) mm, rotated rx -179.9 ry 0 rz -90 deg; joints [36.931, -66.9, 102.332, -126.845, 48.647, 139.509]
  MoveL 1241 to (313.17, 61.67, -154.87) mm, rotated rx -179.9 ry 0 rz -90 deg; joints [36.856, -66.829, 102.238, -126.904, 48.584, 139.533]
  MoveL 1242 to (313.11, 61.6, -157.05) mm, rotated rx -179.9 ry 0 rz -90 deg; joints [36.802, -66.722, 102.091, -126.931, 48.526, 139.527]
  MoveL 1243 to (313.83, 61.52, -159.11) mm, rotated rx -179.9 ry 0 rz -90 deg; joints [36.775, -66.591, 101.911, -126.922, 48.478, 139.491]
  MoveL 1244 to (315.24, 61.44, -160.78) mm, rotated rx -179.9 ry 0 rz -90 deg; joints [36.78, -66.456, 101.722, -126.879, 48.45, 139.43]
  MoveL 1245 to (317.15, 61.37, -161.84) mm, rotated rx -179.9 ry 0 rz -90 deg; joints [36.816, -66.332, 101.548, -126.808, 48.443, 139.354]
  MoveL 1246 to (319.32, 61.29, -162.15) mm, rotated rx -179.9 ry 0 rz -90 deg; joints [36.877, -66.235, 101.414, -126.719, 48.46, 139.273]
  MoveL 1247 to (321.45, 61.21, -161.66) mm, rotated rx -179.9 ry 0 rz -90 deg; joints [36.956, -66.179, 101.336, -126.625, 48.5, 139.199]
  MoveL 1248 to (323.27, 61.14, -160.45) mm, rotated rx -179.9 ry 0 rz -90 deg; joints [37.043, -66.169, 101.326, -126.538, 48.556, 139.142]
  MoveL 1249 to (324.53, 61.06, -158.67) mm, rotated rx -179.9 ry 0 rz -90 deg; joints [37.125, -66.208, 101.386, -126.469, 48.623, 139.111]
  MoveL 1250 to (325.08, 60.98, -156.56) mm, rotated rx -179.9 ry 0 rz -90 deg; joints [37.193, -66.289, 101.507, -126.429, 48.691, 139.11]
  MoveL 1251 to (324.85, 60.91, -154.39) mm, rotated rx -179.9 ry 0 rz -90 deg; joints [37.238, -66.402, 101.674, -126.423, 48.753, 139.139]
  MoveL 1252 to (323.85, 60.83, -152.44) mm, rotated rx -179.9 ry 0 rz -90 deg; joints [37.253, -66.532, 101.866, -126.451, 48.8, 139.196]
  MoveL 1253 to (322.23, 60.75, -150.98) mm, rotated rx -179.9 ry 0 rz -90 deg; joints [37.237, -66.661, 102.058, -126.511, 48.827, 139.273]
  MoveL 1254 to (320.19, 60.68, -150.19) mm, rotated rx -179.9 ry 0 rz -90 deg; joints [37.192, -66.773, 102.225, -126.596, 48.83, 139.361]
  MoveL 1255 to (318, 60.6, -150.18) mm, rotated rx -179.9 ry 0 rz -90 deg; joints [37.123, -66.851, 102.345, -126.694, 48.809, 139.45]
  MoveL 1256 to (315.96, 60.52, -150.95) mm, rotated rx -179.9 ry 0 rz -90 deg; joints [37.039, -66.887, 102.403, -126.795, 48.769, 139.529]
  MoveL 1257 to (314.32, 60.45, -152.39) mm, rotated rx -179.9 ry 0 rz -90 deg; joints [36.952, -66.873, 102.392, -126.884, 48.713, 139.587]
  MoveL 1258 to (313.31, 60.37, -154.33) mm, rotated rx -179.9 ry 0 rz -90 deg; joints [36.874, -66.813, 102.314, -126.951, 48.651, 139.619]
  MoveL 1259 to (313.05, 60.29, -156.5) mm, rotated rx -179.9 ry 0 rz -90 deg; joints [36.814, -66.714, 102.179, -126.986, 48.591, 139.621]
  MoveL 1260 to (313.58, 60.22, -158.62) mm, rotated rx -179.9 ry 0 rz -90 deg; joints [36.78, -66.588, 102.005, -126.987, 48.54, 139.591]
  MoveL 1261 to (314.83, 60.14, -160.41) mm, rotated rx -179.9 ry 0 rz -90 deg; joints [36.777, -66.452, 101.815, -126.952, 48.506, 139.536]
  MoveL 1262 to (316.64, 60.06, -161.64) mm, rotated rx -179.9 ry 0 rz -90 deg; joints [36.805, -66.324, 101.636, -126.887, 48.493, 139.463]
  MoveL 1263 to (318.76, 59.99, -162.14) mm, rotated rx -179.9 ry 0 rz -90 deg; joints [36.86, -66.219, 101.489, -126.802, 48.504, 139.382]
  MoveL 1264 to (320.93, 59.91, -161.86) mm, rotated rx -179.9 ry 0 rz -90 deg; joints [36.936, -66.152, 101.396, -126.707, 48.538, 139.306]
  MoveL 1265 to (322.85, 59.83, -160.82) mm, rotated rx -179.9 ry 0 rz -90 deg; joints [37.021, -66.13, 101.369, -126.617, 48.591, 139.244]
  MoveL 1266 to (324.28, 59.76, -159.16) mm, rotated rx -179.9 ry 0 rz -90 deg; joints [37.106, -66.157, 101.411, -126.543, 48.656, 139.206]
  MoveL 1267 to (325.02, 59.68, -157.11) mm, rotated rx -179.9 ry 0 rz -90 deg; joints [37.179, -66.228, 101.518, -126.495, 48.724, 139.197]
  MoveL 1268 to (324.98, 59.6, -154.92) mm, rotated rx -179.9 ry 0 rz -90 deg; joints [37.23, -66.334, 101.675, -126.48, 48.789, 139.218]
  MoveL 1269 to (324.17, 59.53, -152.89) mm, rotated rx -179.9 ry 0 rz -90 deg; joints [37.253, -66.461, 101.863, -126.499, 48.84, 139.269]
  MoveL 1270 to (322.68, 59.45, -151.29) mm, rotated rx -179.9 ry 0 rz -90 deg; joints [37.245, -66.592, 102.058, -126.552, 48.872, 139.341]
  MoveL 1271 to (320.73, 59.37, -150.32) mm, rotated rx -179.9 ry 0 rz -90 deg; joints [37.207, -66.71, 102.233, -126.631, 48.882, 139.428]
  MoveL 1272 to (318.55, 59.3, -150.11) mm, rotated rx -179.9 ry 0 rz -90 deg; joints [37.143, -66.798, 102.366, -126.727, 48.867, 139.517]
  MoveL 1273 to (316.45, 59.22, -150.68) mm, rotated rx -179.9 ry 0 rz -90 deg; joints [37.062, -66.845, 102.441, -126.828, 48.831, 139.599]
  MoveL 1274 to (314.68, 59.14, -151.97) mm, rotated rx -179.9 ry 0 rz -90 deg; joints [36.975, -66.844, 102.448, -126.921, 48.779, 139.664]
  MoveL 1275 to (313.49, 59.07, -153.81) mm, rotated rx -179.9 ry 0 rz -90 deg; joints [36.893, -66.795, 102.386, -126.995, 48.718, 139.703]
  MoveL 1276 to (313.04, 58.99, -155.95) mm, rotated rx -179.9 ry 0 rz -90 deg; joints [36.827, -66.705, 102.264, -127.039, 48.656, 139.712]
  MoveL 1277 to (313.37, 58.91, -158.1) mm, rotated rx -179.9 ry 0 rz -90 deg; joints [36.786, -66.584, 102.098, -127.049, 48.602, 139.691]
  MoveL 1278 to (314.45, 58.84, -160) mm, rotated rx -179.9 ry 0 rz -90 deg; joints [36.775, -66.449, 101.91, -127.022, 48.563, 139.641]
  MoveL 1279 to (316.14, 58.76, -161.39) mm, rotated rx -179.9 ry 0 rz -90 deg; joints [36.796, -66.317, 101.725, -126.964, 48.545, 139.572]
  MoveL 1280 to (318.21, 58.68, -162.09) mm, rotated rx -179.9 ry 0 rz -90 deg; joints [36.845, -66.205, 101.568, -126.883, 48.55, 139.492]
  MoveL 1281 to (320.39, 58.61, -162) mm, rotated rx -179.9 ry 0 rz -90 deg; joints [36.916, -66.127, 101.46, -126.79, 48.578, 139.413]
  MoveL 1282 to (322.4, 58.53, -161.14) mm, rotated rx -179.9 ry 0 rz -90 deg; joints [37, -66.094, 101.416, -126.697, 48.627, 139.346]
  MoveL 1283 to (323.98, 58.45, -159.63) mm, rotated rx -179.9 ry 0 rz -90 deg; joints [37.086, -66.108, 101.44, -126.618, 48.689, 139.302]
  MoveL 1284 to (324.9, 58.37, -157.65) mm, rotated rx -179.9 ry 0 rz -90 deg; joints [37.163, -66.169, 101.532, -126.563, 48.758, 139.285]
  MoveL 1285 to (325.07, 58.3, -155.47) mm, rotated rx -179.9 ry 0 rz -90 deg; joints [37.22, -66.268, 101.678, -126.539, 48.824, 139.299]
  MoveL 1286 to (324.44, 58.22, -153.38) mm, rotated rx -179.9 ry 0 rz -90 deg; joints [37.251, -66.391, 101.861, -126.549, 48.879, 139.343]
  MoveL 1287 to (323.11, 58.14, -151.64) mm, rotated rx -179.9 ry 0 rz -90 deg; joints [37.251, -66.522, 102.056, -126.594, 48.917, 139.41]
  MoveL 1288 to (321.25, 58.07, -150.49) mm, rotated rx -179.9 ry 0 rz -90 deg; joints [37.22, -66.645, 102.238, -126.667, 48.932, 139.494]
  MoveL 1289 to (319.11, 57.99, -150.09) mm, rotated rx -179.9 ry 0 rz -90 deg; joints [37.162, -66.741, 102.384, -126.76, 48.924, 139.584]
  MoveL 1290 to (316.96, 57.91, -150.47) mm, rotated rx -179.9 ry 0 rz -90 deg; joints [37.084, -66.799, 102.475, -126.861, 48.893, 139.669]
  MoveL 1291 to (315.08, 57.84, -151.59) mm, rotated rx -179.9 ry 0 rz -90 deg; joints [36.997, -66.811, 102.499, -126.958, 48.845, 139.739]
  MoveL 1292 to (313.73, 57.76, -153.31) mm, rotated rx -179.9 ry 0 rz -90 deg; joints [36.913, -66.774, 102.454, -127.037, 48.785, 139.785]
  MoveL 1293 to (313.08, 57.68, -155.39) mm, rotated rx -179.9 ry 0 rz -90 deg; joints [36.842, -66.693, 102.346, -127.089, 48.723, 139.802]
  MoveL 1294 to (313.21, 57.61, -157.57) mm, rotated rx -179.9 ry 0 rz -90 deg; joints [36.794, -66.579, 102.189, -127.108, 48.666, 139.788]
  MoveL 1295 to (314.12, 57.53, -159.56) mm, rotated rx -179.9 ry 0 rz -90 deg; joints [36.776, -66.446, 102.004, -127.091, 48.622, 139.745]
  MoveL 1296 to (315.67, 57.45, -161.1) mm, rotated rx -179.9 ry 0 rz -90 deg; joints [36.788, -66.312, 101.816, -127.04, 48.598, 139.68]
  MoveL 1297 to (317.67, 57.38, -161.99) mm, rotated rx -179.9 ry 0 rz -90 deg; joints [36.831, -66.193, 101.65, -126.964, 48.597, 139.601]
  MoveL 1298 to (319.85, 57.3, -162.1) mm, rotated rx -179.9 ry 0 rz -90 deg; joints [36.897, -66.106, 101.528, -126.872, 48.62, 139.521]
  MoveL 1299 to (321.93, 57.22, -161.43) mm, rotated rx -179.9 ry 0 rz -90 deg; joints [36.979, -66.06, 101.467, -126.778, 48.663, 139.45]
  MoveL 1300 to (323.63, 57.15, -160.06) mm, rotated rx -179.9 ry 0 rz -90 deg; joints [37.065, -66.063, 101.474, -126.694, 48.723, 139.399]
  MoveL 1301 to (324.74, 57.07, -158.18) mm, rotated rx -179.9 ry 0 rz -90 deg; joints [37.146, -66.112, 101.549, -126.632, 48.79, 139.375]
  MoveL 1302 to (325.1, 56.99, -156.02) mm, rotated rx -179.9 ry 0 rz -90 deg; joints [37.209, -66.202, 101.683, -126.599, 48.858, 139.382]
  MoveL 1303 to (324.67, 56.92, -153.88) mm, rotated rx -179.9 ry 0 rz -90 deg; joints [37.247, -66.321, 101.859, -126.601, 48.917, 139.418]
  MoveL 1304 to (323.51, 56.84, -152.03) mm, rotated rx -179.9 ry 0 rz -90 deg; joints [37.254, -66.452, 102.053, -126.638, 48.96, 139.48]
  MoveL 1305 to (321.76, 56.76, -150.72) mm, rotated rx -179.9 ry 0 rz -90 deg; joints [37.231, -66.578, 102.241, -126.704, 48.981, 139.561]
  MoveL 1306 to (319.66, 56.69, -150.11) mm, rotated rx -179.9 ry 0 rz -90 deg; joints [37.179, -66.682, 102.398, -126.793, 48.979, 139.65]
  MoveL 1307 to (317.48, 56.61, -150.3) mm, rotated rx -179.9 ry 0 rz -90 deg; joints [37.106, -66.751, 102.504, -126.894, 48.954, 139.738]
  MoveL 1308 to (315.51, 56.53, -151.24) mm, rotated rx -179.9 ry 0 rz -90 deg; joints [37.02, -66.775, 102.546, -126.992, 48.909, 139.812]
  MoveL 1309 to (314.01, 56.46, -152.83) mm, rotated rx -179.9 ry 0 rz -90 deg; joints [36.934, -66.75, 102.518, -127.077, 48.852, 139.865]
  MoveL 1310 to (313.17, 56.38, -154.85) mm, rotated rx -179.9 ry 0 rz -90 deg; joints [36.859, -66.679, 102.425, -127.137, 48.789, 139.889]
  MoveL 1311 to (313.11, 56.3, -157.03) mm, rotated rx -179.9 ry 0 rz -90 deg; joints [36.805, -66.572, 102.278, -127.165, 48.73, 139.883]
  MoveL 1312 to (313.82, 56.23, -159.09) mm, rotated rx -179.9 ry 0 rz -90 deg; joints [36.778, -66.443, 102.098, -127.156, 48.683, 139.847]
  MoveL 1313 to (315.23, 56.15, -160.77) mm, rotated rx -179.9 ry 0 rz -90 deg; joints [36.783, -66.307, 101.909, -127.114, 48.653, 139.786]
  MoveL 1314 to (317.13, 56.07, -161.83) mm, rotated rx -179.9 ry 0 rz -90 deg; joints [36.818, -66.183, 101.735, -127.043, 48.646, 139.71]
  MoveL 1315 to (319.3, 56, -162.15) mm, rotated rx -179.9 ry 0 rz -90 deg; joints [36.879, -66.087, 101.6, -126.954, 48.663, 139.63]
  MoveL 1316 to (321.43, 55.92, -161.67) mm, rotated rx -179.9 ry 0 rz -90 deg; joints [36.958, -66.03, 101.522, -126.86, 48.701, 139.555]
  MoveL 1317 to (323.25, 55.84, -160.46) mm, rotated rx -179.9 ry 0 rz -90 deg; joints [37.045, -66.02, 101.512, -126.772, 48.757, 139.499]
  MoveL 1318 to (324.53, 55.77, -158.69) mm, rotated rx -179.9 ry 0 rz -90 deg; joints [37.127, -66.058, 101.57, -126.703, 48.823, 139.467]
  MoveL 1319 to (325.08, 55.69, -156.58) mm, rotated rx -179.9 ry 0 rz -90 deg; joints [37.195, -66.139, 101.691, -126.663, 48.892, 139.466]
  MoveL 1320 to (324.85, 55.61, -154.4) mm, rotated rx -179.9 ry 0 rz -90 deg; joints [37.24, -66.251, 101.858, -126.656, 48.954, 139.495]
  MoveL 1321 to (323.86, 55.54, -152.46) mm, rotated rx -179.9 ry 0 rz -90 deg; joints [37.256, -66.381, 102.05, -126.683, 49.001, 139.551]
  MoveL 1322 to (322.24, 55.46, -150.99) mm, rotated rx -179.9 ry 0 rz -90 deg; joints [37.24, -66.51, 102.242, -126.743, 49.029, 139.628]
  MoveL 1323 to (320.21, 55.38, -150.19) mm, rotated rx -179.9 ry 0 rz -90 deg; joints [37.195, -66.621, 102.409, -126.827, 49.033, 139.716]
  MoveL 1324 to (318.02, 55.31, -150.18) mm, rotated rx -179.9 ry 0 rz -90 deg; joints [37.126, -66.7, 102.529, -126.926, 49.013, 139.805]
  MoveL 1325 to (315.98, 55.23, -150.94) mm, rotated rx -179.9 ry 0 rz -90 deg; joints [37.043, -66.735, 102.588, -127.026, 48.973, 139.884]
  MoveL 1326 to (314.33, 55.15, -152.38) mm, rotated rx -179.9 ry 0 rz -90 deg; joints [36.956, -66.723, 102.578, -127.116, 48.918, 139.942]
  MoveL 1327 to (313.31, 55.08, -154.31) mm, rotated rx -179.9 ry 0 rz -90 deg; joints [36.877, -66.663, 102.5, -127.183, 48.856, 139.974]
